Omron Sysmac Studio project Auto Connect Project (Sysmac Studio 1.66.0.64007, StandardProject)

# Controller new_Controller_0: NX502-1300 version 1.69
Units and slaves: Node9 : CPX-AP-A-EC-M12(E007); 0 : CPX-AP-A-EC-M12(M1); 1 : CPX-AP-A-16DI-D-M12-5P(M2); 2 : CPX-AP-A-16DI-D-M12-5P(M3); 3 : VABX-A-P-EL-E12-APA(M4); Node10 : NXR-ILM08C-ECT (E006); Unit 1 : NX-PF0730 (N1); Unit 3 : NX-SID800 (N3); Unit 4 : NX-SID800 (N4); Unit 5 : NX-SID800 (N5); Unit 6 : NX-SOD400 (N6); Unit 7 : NX-SOD400 (N7); Unit 8 : NX-PD1000 (N8); Unit 9 : NX-ID5442 (N9); Unit 10 : NX-ID5442 (N10); Unit 11 : NX-OD5256 (N11); Unit 12 : NX-OD5256 (N12)
Axis SC1501Ax, settings changed from default: AxisType=ServoType, UnitsConversion=EnumElement2, UnitsNumerator=8388608, ReducerUse=EnumElement2, UnitsDenominator=12.5, TravelDistancePerWorkRotation=125, MotorGearRatio=7, MaxVelocity=3199, MaxJogVelocity=3199, HomingMode=BackupAndPressingTime, StartDirection=NegativeDirection, OriginInputDetectionDirection=NegativeDirection, HomingVelocity=20, HomingApproachVelocity=20, HomingAcceleration=10, HomingJerk=10, PushTime=0, CompensationVelocity=20, EncoderTypes=Abs
Axis SC2301Ax, settings changed from default: AxisNumber=1, AxisType=ServoType, UnitsConversion=EnumElement2, UnitsNumerator=8601600, UnitsDenominator=30.0372, TravelDistancePerWorkRotation=300.37, MotorGearRatio=10, MaxVelocity=7499, MaxJogVelocity=7499, MaxAcceleration=10000, MaxDeceleration=10000, FollowingErrorLimit=500, FollowingErrorAlarmLimit=500, HomingMode=BackupAndPressingTime, HomingVelocity=10, HomingApproachVelocity=10, HomingAcceleration=50, HomingDeceleration=50, HomingJerk=100, PushTime=0
Axis SC2302Ax, settings changed from default: AxisNumber=2, AxisType=ServoType, UnitsConversion=EnumElement2, UnitsNumerator=8388608, ReducerUse=EnumElement2, UnitsDenominator=30.0372, TravelDistancePerWorkRotation=300.37, MotorGearRatio=10, MaxVelocity=7499, MaxJogVelocity=7499, MaxAcceleration=10000, MaxDeceleration=10000, FollowingErrorLimit=500, FollowingErrorAlarmLimit=500, HomingMode=BackupAndPressingTime, StartDirection=NegativeDirection, OriginInputDetectionDirection=NegativeDirection, HomingVelocity=10, HomingApproachVelocity=10, HomingAcceleration=50, HomingDeceleration=50, HomingJerk=50, PushTime=0
Axis SC2303Ax, settings changed from default: AxisNumber=3, AxisType=ServoType, UnitsConversion=EnumElement2, UnitsNumerator=8388608, ReducerUse=EnumElement2, UnitsDenominator=30.0372, TravelDistancePerWorkRotation=300.37, MotorGearRatio=10, MaxVelocity=7499, MaxJogVelocity=7499, MaxAcceleration=10000, MaxDeceleration=10000, FollowingErrorLimit=500, FollowingErrorAlarmLimit=500, HomingMode=BackupAndPressingTime, StartDirection=NegativeDirection, OriginInputDetectionDirection=NegativeDirection, HomingVelocity=10, HomingApproachVelocity=10, HomingAcceleration=50, HomingJerk=50, PushTime=0
Axis SC6401Ax, settings changed from default: AxisNumber=4, AxisType=ServoType, UnitsConversion=EnumElement2, UnitsNumerator=8388608, ReducerUse=EnumElement2, UnitsDenominator=9, TravelDistancePerWorkRotation=125, MotorGearRatio=10, MaxVelocity=2299, MaxJogVelocity=2299, HomingMode=BackupAndProximitySignalOn, StartDirection=NegativeDirection, OriginInputDetectionDirection=NegativeDirection, HomingVelocity=20, HomingApproachVelocity=20, EncoderTypes=Abs
Task PrimaryTask (priority 4, period or condition 4000): Control, Inputs, Outputs
Library OneS_monitor 1.0.0 (contents left out)

TYPE CylinderD : STRUCT
    AutoExtend : BOOL;
    AutoRetract : BOOL;
    ManExtend : BOOL;
    ManRetract : BOOL;
    ManOff : BOOL;
    ForceExtend : BOOL;
    ForceRetract : BOOL;
    ExtendSol : BOOL;
    RetractSol : BOOL;
    TestCycleSelect : BOOL;
    AlarmMute : BOOL;
    ExtendReed : BOOL;
    RetractReed : BOOL;
    Alarm : BOOL;
    CountReset : BOOL;
    CycleExtendTime : LREAL;
    CycleRetractTime : LREAL;
    ExtendTime : LREAL;
    RetractTime : LREAL;
    ExtendTimeAcc : LREAL;
    RetractTimeAcc : LREAL;
    AlarmCode : DINT;
    ManualCode : DINT;
    ExtendReedsUsed : DINT;
    RetractReedsUsed : DINT;
    ExtendCount : DINT;
    RetractCount : DINT;
    TagName : STRING[256];
    TagDescription : STRING[256];
    ErrorTrigger : ARRAY[0..19] OF BOOL;
    ManualTrigger : ARRAY[0..19] OF BOOL;
END_STRUCT END_TYPE
TYPE MotorD : STRUCT
    AlarmMute : BOOL;
    AutoForward : BOOL;
    ManForward : BOOL;
    ManReverse : BOOL;
    ManOFF : BOOL;
    AutoReverse : BOOL;
    ForceFoward : BOOL;
    ForceReverse : BOOL;
    RunFeedback : BOOL;
    Alarm : BOOL;
    ForceOFF : BOOL;
    CountReset : BOOL;
    ManualCode : DINT;
    AlarmCode : DINT;
    RunCount : DINT;
    RunHours : REAL;
    Faulttime : LREAL;
    FaulttimeAcc : LREAL;
    TagName : STRING[256];
    TagDescription : STRING[256];
    ErrorTrigger : ARRAY[0..19] OF BOOL;
    ManualTrigger : ARRAY[0..19] OF BOOL;
END_STRUCT END_TYPE
TYPE MotorVSDD : STRUCT
    AlarmMute : BOOL;
    AutoForward : BOOL;
    ManForward : BOOL;
    ManReverse : BOOL;
    ManOFF : BOOL;
    AutoReverse : BOOL;
    ForceFoward : BOOL;
    ForceReverse : BOOL;
    ForceOFF : BOOL;
    CountReset : BOOL;
    RunFeedback : BOOL;
    ManualCode : DINT;
    AlarmCode : DINT;
    RunCount : DINT;
    RunHours : REAL;
    Faulttime : LREAL;
    FaulttimeAcc : LREAL;
    AutoSpeed : UINT;
    ManualSpeed : UINT;
    Speed : UINT;
    Alarm : BOOL;
    TagName : STRING[256];
    TagDescription : STRING[256];
    ErrorTrigger : ARRAY[0..19] OF BOOL;
    ManualTrigger : ARRAY[0..19] OF BOOL;
END_STRUCT END_TYPE
TYPE ServoD : STRUCT
    JogForward : BOOL;
    JogReverse : BOOL;
    JogToPosition : BOOL;
    ManualHome : BOOL;
    AutoHome : BOOL;
    Homed : BOOL;
    Alarm : BOOL;
    Enabled : BOOL;
    AxisErrorCode : WORD;
    RunHours : REAL;
    JogSpeed : LREAL;
    JogAccel : LREAL;
    JogDecel : LREAL;
    JogPos : LREAL;
    JogJerk : LREAL;
    JogType : DINT;
    ActualPos : LREAL;
    ActualVel : LREAL;
    PowerEnable : BOOL;
    MovePos1 : BOOL;
    Pos1 : LREAL;
    Pos1Vel : LREAL;
    Pos1Accel : LREAL;
    Pos1Decel : LREAL;
    Pos1Jerk : LREAL;
    Pos1Movetype : DINT;
    Pos1OK : BOOL;
    MovePos2 : BOOL;
    Pos2 : LREAL;
    Pos2Vel : LREAL;
    Pos2Accel : LREAL;
    Pos2Decel : LREAL;
    Pos2Jerk : LREAL;
    Pos2Movetype : DINT;
    Pos2OK : BOOL;
    MovePos3 : BOOL;
    Pos3 : LREAL;
    Pos3Vel : LREAL;
    Pos3Accel : LREAL;
    Pos3Decel : LREAL;
    Pos3Jerk : LREAL;
    Pos3Movetype : DINT;
    Pos3OK : BOOL;
    MovePos4 : BOOL;
    Pos4 : LREAL;
    Pos4Vel : LREAL;
    Pos4Accel : LREAL;
    Pos4Decel : LREAL;
    Pos4Jerk : LREAL;
    Pos4OK : BOOL;
    Pos4Movetype : DINT;
    MovePos5 : BOOL;
    Pos5 : LREAL;
    Pos5Vel : LREAL;
    Pos5Accel : LREAL;
    Pos5Decel : LREAL;
    Pos5OK : BOOL;
    Pos5Movetype : DINT;
    Pos5Jerk : LREAL;
    MoveVelSpeed : LREAL;
    MovePos6 : BOOL;
    Pos6 : LREAL;
    Pos6Vel : LREAL;
    Pos6Accel : LREAL;
    Pos6Decel : LREAL;
    Pos6Jerk : LREAL;
    Pos6OK : BOOL;
    Pos6Movetype : DINT;
    MoveVel : BOOL;
    MoveVelAcc : LREAL;
    MoveVeldec : LREAL;
    MoveVelJerk : LREAL;
    MoveVelType : DINT;
    MoveVelCon : BOOL;
    MoveVelOK : BOOL;
    PositionTolerence : LREAL;
    AlarmCode : DWORD;
    ManualCode : DINT;
    TagName : STRING[256];
    TagDescription : STRING[256];
    ErrorTrigger : ARRAY[0..19] OF BOOL;
    ManualTrigger : ARRAY[0..19] OF BOOL;
END_STRUCT END_TYPE
TYPE MiscInD : STRUCT
    ManOn : BOOL;
    ManOff : BOOL;
    ForceOn : BOOL;
    ForceOff : BOOL;
    Fault : BOOL;
    InputFault : BOOL;
    Mute : BOOL;
    Value : BOOL;
    Input : BOOL;
    AlarmCode : DINT;
    Alarm : BOOL;
    ManualCode : DINT;
    DebounceOFFtime : LREAL;
    DebounceONtime : LREAL;
    FaultTime : LREAL;
    AccumulatedOnTime : LREAL;
    AccumulatedOffTime : LREAL;
    FaultAccumulatedTime : LREAL;
    TagName : STRING[256];
    TagDescription : STRING[256];
    ErrorTrigger : ARRAY[0..19] OF BOOL;
    ManualTrigger : ARRAY[0..19] OF BOOL;
END_STRUCT END_TYPE
TYPE MiscOutD : STRUCT
    ManOn : BOOL;
    ManOff : BOOL;
    ForceOn : BOOL;
    ForceOff : BOOL;
    Fault : BOOL;
    Mute : BOOL;
    Value : BOOL;
    Auto : BOOL;
    AlarmCode : DINT;
    ManualCode : DINT;
    FaultTime : LREAL;
    FaultAccumulatedTime : LREAL;
    Alarm : BOOL;
    TagName : STRING[256];
    TagDescription : STRING[256];
    ErrorTrigger : ARRAY[0..19] OF BOOL;
    ManualTrigger : ARRAY[0..19] OF BOOL;
END_STRUCT END_TYPE
TYPE SequenceD : STRUCT
    CurrentStep : ARRAY[0..31] OF BOOL;
    StepTime : ARRAY[0..31] OF REAL;
    StepTimeAcc : REAL;
    Matrix : ARRAY[0..31] OF Dint_Bool;
    Matrix_In : ARRAY[0..31] OF DINT;
    Outputs : ARRAY[0..0] OF Dint_Bool;
    StepReq : DINT;
    StepNum : DINT;
    StepPrev : DINT;
    LastActiveStep : DINT;
    StepTimeDn : BOOL;
    History : ARRAY[0..9] OF SequenceHistory;
    SequenceDisabled : BOOL;
    TagName : STRING[256];
    TagDiscription : STRING[256];
    LocalMessageOffset : DINT;
    LocalMessageValue : DINT;
    Flag : ARRAY[0..9] OF BOOL;
    DeviceAlarm : BOOL;
    Held : BOOL;
    Stopped : BOOL;
    Homed : BOOL;
    TagName_Copy : STRING[256];
    TagDescription : STRING[256];
END_STRUCT END_TYPE
TYPE SequenceHistory : STRUCT
    Num : DINT;
    Messageoffset : DINT;
    ElapsedTime : REAL;
END_STRUCT END_TYPE
TYPE System : STRUCT
    ScanRate : REAL;
    Alarm : BOOL;
    Alarm_Ack : BOOL;
    Energized : BOOL;
    Safetyresetselect : BOOL;
    CurrentStep : DINT;
    ResetSelect : BOOL;
    Messages : DINT;
    AlertMessages : DINT;
    SafetyMessages : DINT;
    HomeSelect : BOOL;
    HomeEnabled : BOOL;
    Homed : BOOL;
    StartSelect : BOOL;
    HoldSelect : BOOL;
    Alarm_AckSelect : BOOL;
    StopSelect : BOOL;
    Alert : BOOL;
    CycleTime : LREAL;
    ShippersPerMin : LREAL;
    TotalRunHours : LREAL;
    CartonsPerMin : LREAL;
END_STRUCT END_TYPE
TYPE TrackTrace : STRUCT
    Carton : DINT;
    Booklet : BOOL;
END_STRUCT END_TYPE
TYPE Vis_In : STRUCT
    InfoBits : SINT;
    Reserved1 : SINT;
    Congiguration_change_device : SINT;
    Reserved2 : BYTE;
    Device_Status : Device_status;
    Fault_code : DINT;
    Counters : ARRAY[0..5] OF DINT;
    Read_Cyc_report : ARRAY[0..3] OF int;
    Decode_Cyc_report : ARRAY[0..3] OF int;
    CodeType : DINT;
    PixelPerElement : real;
    Decode_length : DINT;
    Decode_data : ARRAY[0..435] OF Byte;
END_STRUCT END_TYPE
TYPE Device_status : STRUCT
    Run_mode : BOOL;  (* offset 0.0 *)
    Triger_Acknowledged : BOOL;  (* offset 0.1 *)
    Exposure_done : BOOL;  (* offset 0.2 *)
    Decoding : BOOL;  (* offset 0.3 *)
    Data_is_Ready : BOOL;  (* offset 0.4 *)
    Read_cyc_pass : BOOL;  (* offset 0.5 *)
    Read_cyc_fail : BOOL;  (* offset 0.6 *)
    General_Fault : BOOL;  (* offset 0.7 *)
    New_match_code_acknowledged : BOOL;  (* offset 1.0 *)
    Match_code_enabled : BOOL;  (* offset 1.1 *)
    Image_sensor_Calibrating : BOOL;  (* offset 1.2 *)
    Image_sensor_Calibrating_complete : BOOL;  (* offset 1.3 *)
    Training : BOOL;  (* offset 1.4 *)
    Training_complete : BOOL;  (* offset 1.5 *)
    Optimizing_complete : BOOL;  (* offset 1.6 *)
    Auto_image_photometry_enabled : BOOL;  (* offset 1.7 *)
    Auto_image_photometry_Complete : BOOL;  (* offset 2.0 *)
    Output1_Status : BOOL;  (* offset 2.1 *)
    Output2_Status : BOOL;  (* offset 2.2 *)
    Output3_Status : BOOL;  (* offset 2.3 *)
    Buffer_overflow : BOOL;  (* offset 2.4 *)
    Reserved : ARRAY[0..9] OF Bool;  (* offset 2.5 *)
END_STRUCT END_TYPE
TYPE Vis_out : STRUCT
    Command : commands;
END_STRUCT END_TYPE
TYPE commands : STRUCT
    Run_mode : BOOL;  (* offset 0.0 *)
    Trigger : BOOL;  (* offset 0.1 *)
    Enable_match_code : BOOL;  (* offset 0.2 *)
    Reset_general_fault : BOOL;  (* offset 0.3 *)
    Clear_NoRead_CycRead_Count : BOOL;  (* offset 0.4 *)
    Clear_Mismatch_CycRead_Count : BOOL;  (* offset 0.5 *)
    Clear_NoRead_Count : BOOL;  (* offset 0.6 *)
    Clear_trigger_Count : BOOL;  (* offset 0.7 *)
    Clear_MatchCode_count : BOOL;  (* offset 1.0 *)
    Clear_Mismatch_Count : BOOL;  (* offset 1.1 *)
    Output_1 : BOOL;  (* offset 1.2 *)
    Output_2 : BOOL;  (* offset 1.3 *)
    Output_3 : BOOL;  (* offset 1.4 *)
    Reserved : ARRAY[0..17] OF Bool;  (* offset 1.5 *)
END_STRUCT END_TYPE
TYPE Resulted : STRUCT
    ScanData : STRING[32];
    Done : BOOL;
    Match : BOOL;
    Mismatch : BOOL;
    Alarm : BOOL;
END_STRUCT END_TYPE
TYPE ScannerD : STRUCT
    Result : Resulted;
    ExpectedCode : STRING[32];
    Trigger : BOOL;
    Alarm : BOOL;
    AlarmMute : BOOL;
    AlarmCode : DINT;
END_STRUCT END_TYPE
TYPE BatchDetails : STRUCT
    Start : BOOL;  (* Batch Start *)
    Running : BOOL;  (* Running *)
    Innitiate : BOOL;  (* Innitialization *)
    Complete : BOOL;  (* Batch Complete *)
    Goodshippers : REAL;  (* Good shipper *)
    Rejectshippers : REAL;  (* Reject shipper *)
    Totalshippers : REAL;  (* Total shipper *)
END_STRUCT END_TYPE
TYPE RecipeD : STRUCT
    RealValue : ARRAY[0..49] OF REAL;
    MechValue : ARRAY[0..49] OF REAL;
END_STRUCT END_TYPE
TYPE Word_Bool : UNION
    Word_value : Word;
    Bool_value : ARRAY[0..31] OF BOOL;
END_UNION END_TYPE
TYPE Dint_Bool : UNION
    Dint_Value : DWORD;
    Bool_Value : ARRAY[0..31] OF BOOL;
END_UNION END_TYPE

VAR_GLOBAL RETAIN
    CY1601 : CylinderD;  (* Shipper Support Cylinder; published *)
    PE1404 : MiscInD;  (* published *)
    CY2502 : CylinderD;  (* Product Clamp CYL 2; published *)
    CY2501 : CylinderD;  (* Vertical CYL 1; published *)
    CY2402 : CylinderD;  (* Vertical Stopper CYL; published *)
    CY2401 : CylinderD;  (* Matrix Pusher CYL; published *)
    CY2302 : CylinderD;  (* Matrix Side Shift Cyl 1 at matrix area 2; published *)
    CY2303 : CylinderD;  (* Bottles stopper Cyl 1 @ area 1; RetractReed Bottles stopper Cyl 1 @ area 1; published *)
    CY2301 : CylinderD;  (* Matrix Side Shift Cyl 1 at matrix area 1; published *)
    PE1501 : MiscInD;  (* Shipper Presence Detect; Value Plucker Head Shipper Presence Detect; published *)
    PE2201 : MiscInD;  (* Shipper Squaring Detect PE; published *)
    PE2202 : MiscInD;  (* Bottom tape Low level Detect; published *)
    PE2203 : MiscInD;  (* Bottom Tape apply Check PE 1; published *)
    PE2301 : MiscInD;  (* Matrix Present Detetct Eye1; published *)
    PE2302 : MiscInD;  (* Matrix Present Detetct Eye2; published *)
    PE2303 : MiscInD;  (* Product Presnt @ Collation Entrc; published *)
    PE2401 : MiscInD;  (* Matrix Present Detect; published *)
    PE3401 : MiscInD;  (* Pre-Lable Trigger PE; published *)
    PE3402 : MiscInD;  (* Shipper presence for Palletizer; published *)
    PE6901 : MiscInD;  (* Pallet 1 Presence PE 1; published *)
    PE6902 : MiscInD;  (* Pallet 1 Presence PE 2; published *)
    DI3511 : MiscInD;  (* Pre-Printing Applicator Machine Run Signal; published *)
    DI3501 : MiscInD;  (* Label Applicator Machine Run Signal; published *)
    DI3502 : MiscInD;  (* Label Applicator Machine Accept Signal; published *)
    DI3503 : MiscInD;  (* Label Applicator Machine Reject Signal; published *)
END_VAR
VAR_GLOBAL
    SC2701 : ServoD;  (* Shipper pusher Servo; published *)
END_VAR
VAR_GLOBAL RETAIN
    MO1402 : MotorD;  (* Magazine motor 2; published *)
    MO2301 : MotorD;  (* Infeed Collation Conveyor Motor; published *)
    MO2201 : MotorD;  (* Tapping Machine RH Motor; published *)
    MO2202 : MotorD;  (* Tapping Machine LH Motor; published *)
    IL0302 : MiscOutD;  (* Alert Indication (Amber); published *)
    IL0303 : MiscOutD;  (* Fault Indication (Red); published *)
    DO0301 : MiscOutD;  (* Drives Fault Reset; published *)
    DO3301 : MiscOutD;  (* Aggrigation System Trigger Signal; published *)
    DO3302 : MiscOutD;  (* published *)
    SV0401 : MiscOutD;  (* Pneumatic Quick Exhaust Valve; published *)
    SV1501 : MiscOutD;  (* Plucker Vacuum Sov 1; published *)
    SV2301 : MiscOutD;  (* Vaccume SOL; published *)
    SV2501 : MiscOutD;  (* Pickhead Vacuum Sov 1; published *)
    SV2502 : MiscOutD;  (* Pickhead Vacuum Sov 2; published *)
    PS2501 : MiscInD;  (* Robot pickhead pressure switch; published *)
    PS0401 : MiscInD;  (* Presure Switch; published *)
    IL0301 : MiscOutD;  (* Run Indication (Green); published *)
    P23c : SequenceD;  (* Infeed Conveyor 3; published *)
END_VAR
VAR_GLOBAL
    SafetyDeviceReady : BOOL;  (* Emergency and Guard Door Ready; published *)
END_VAR
VAR_GLOBAL RETAIN
    Batch_Report : BatchDetails;  (* published *)
END_VAR
VAR_GLOBAL
    Shipper_Accept : BOOL;
END_VAR
VAR_GLOBAL RETAIN
    CY2304 : CylinderD;  (* Bottles stopper Cyl 1 @ area 2; published *)
END_VAR
VAR_GLOBAL
    Reject_Matrix_Accept : BOOL;
    Carton_Matrix_Accept : BOOL;
    RO4001_I_PalletizingDone : BOOL;
    Palletizing_Done : BOOL;
    Shipper_Reject : BOOL;
    Shipper_Good_Count : BOOL;
    S_CellEnabled : BOOL;
    SKU_Select : DINT;
END_VAR
VAR_GLOBAL RETAIN
    P27 : SequenceD;  (* Case Erector; Flag[0] Plucker At Shipper Pick Pos; published *)
    PE1602 : MiscInD;  (* published *)
END_VAR
VAR_GLOBAL
    TotalLayers : DINT;  (* published *)
    ShippersPerLayer : DINT;  (* published *)
    IPCcheck : BOOL;  (* published *)
    IPCcheckAlarm : BOOL;
    IPCCheck1 : BOOL;  (* published *)
    P22_TapeAlarm : BOOL;  (* published *)
    RO4001_Alarm : BOOL;
    RO4001_ErrorTrigger : ARRAY[0..9] OF BOOL;  (* published *)
END_VAR
VAR_GLOBAL RETAIN
    DO3502 : MiscOutD;  (* published *)
    DO3501 : MiscOutD;  (* published *)
    PE3501 : MiscInD;  (* published *)
    K1301 : MiscOutD;  (* published *)
    PE1403 : MiscInD;  (* Shipper Forming Detect PE 2; published *)
    PE1402 : MiscInD;  (* Shipper Forming Detect PE 1; published *)
    SV2701 : MiscOutD;  (* published *)
    PE6401 : MiscInD;  (* Shipper Presence Detect Eye; published *)
    PE1801 : MiscInD;  (* Product High Level Detect; published *)
    PE1811 : MiscInD;  (* Bundle High level detect; published *)
    PE1812 : MiscInD;  (* Bundle detect @ Clamp; published *)
    PE1701 : MiscInD;  (* Shipper Presence @ Stopper 1; published *)
    PE1702 : MiscInD;  (* Shipper Presence @ Placing Station; published *)
    PE2501 : MiscInD;  (* published *)
    PE2502 : MiscInD;  (* published *)
    PE2503 : MiscInD;  (* published *)
    PE2801 : MiscInD;  (* Layer Board Magazine Low level detect Eye; published *)
    PE2511 : MiscInD;  (* published *)
    PE2521 : MiscInD;  (* published *)
    PE2702 : MiscInD;  (* published *)
    PE2703 : MiscInD;  (* published *)
END_VAR
VAR_GLOBAL
    PE7101 : MiscInD;  (* Shipper Presence Detect; published *)
END_VAR
VAR_GLOBAL RETAIN
    PE3101 : MiscInD;  (* published *)
    PE2512 : MiscInD;  (* published *)
    PE6911 : MiscInD;  (* published *)
    PE6912 : MiscInD;  (* published *)
    SV1502 : MiscOutD;  (* Plucker Vacuum Sov 1; published *)
    SV1503 : MiscOutD;  (* Plucker Vacuum Sov 1; published *)
    SV2511 : MiscOutD;  (* published *)
    SV2512 : MiscOutD;  (* published *)
    SV2521 : MiscOutD;  (* published *)
    SV7101 : MiscOutD;  (* Shipper Vaccume; published *)
    DO320 : MiscOutD;
    DO0320 : MiscOutD;
    DO0350 : MiscOutD;
    CY1502 : CylinderD;  (* Minor Flap close CYL 2; ExtendReed Minor Flap close CYL 2; published *)
    CY1503 : CylinderD;  (* Major Flap close CYL 1; RetractReed Major Flap close CYL 1; published *)
    CY1504 : CylinderD;  (* Major Flap close CYL 2; RetractReed Major Flap close CYL 1; published *)
    CY1811 : CylinderD;  (* Clamp Cyl 1; published *)
    CY1701 : CylinderD;  (* Shipper Stopper Before Loading station.; published *)
    CY1702 : CylinderD;  (* Shipper Stopper at Loading station.; published *)
    CY1703 : CylinderD;  (* Hopper Cylinder; published *)
    CY2521 : CylinderD;  (* published *)
    CY7101 : CylinderD;  (* Shipper Rotation CYL; published *)
    CY7102 : CylinderD;  (* Shipper Puller and Pusher CYL; published *)
    CY3401 : CylinderD;  (* Shipper Stopper CYL; published *)
    CY3402 : CylinderD;  (* Shipper Rejection/ Accepted CYL; published *)
    DI0350 : MiscInD;  (* published *)
    DI7501 : MiscInD;  (* published *)
    DI7502 : MiscInD;  (* published *)
    DI7503 : MiscInD;  (* published *)
    DI3512 : MiscInD;  (* published *)
    DI3513 : MiscInD;  (* published *)
    MO1801 : MotorD;  (* Infeed Conveyor 1 of Loose Bottles Motor; published *)
    MO1811 : MotorD;  (* Infeed Conveyor 2 of Bundle Bottles Motor; published *)
    MO1701 : MotorD;  (* Main Drive Conveyor Motor; published *)
    MO3101 : MotorD;  (* published *)
    SC1501 : ServoD;  (* Plucker Servo; published *)
END_VAR
VAR_GLOBAL
    SC1501_Ax : _sAXIS_REF;
END_VAR
VAR_GLOBAL RETAIN
    SC6401 : ServoD;  (* Box Transfer Servo; published *)
END_VAR
VAR_GLOBAL
    SC6401_Ax : _sAXIS_REF;
END_VAR
VAR_GLOBAL RETAIN
    SC2301 : ServoD;  (* published *)
END_VAR
VAR_GLOBAL
    SC2301_Ax : _sAXIS_REF;
END_VAR
VAR_GLOBAL RETAIN
    SC2302 : ServoD;  (* published *)
END_VAR
VAR_GLOBAL
    SC2302_Ax : _sAXIS_REF;
END_VAR
VAR_GLOBAL RETAIN
    SC2303 : ServoD;  (* published *)
END_VAR
VAR_GLOBAL
    SC2303_Ax : _sAXIS_REF;
    XC0301_6_I : ARRAY[0..15] OF BOOL;  (* Input Card 1; at IOBus://unit#9/Input Bit 16 bits *)
    XC0301_7_I : ARRAY[0..15] OF BOOL;  (* Input Card 2; at IOBus://unit#10/Input Bit 16 bits *)
END_VAR
VAR_GLOBAL RETAIN
    PS2502 : MiscInD;  (* published *)
END_VAR
VAR_GLOBAL
    XC0301_8_O : ARRAY[0..15] OF BOol;  (* Output Card 1; at IOBus://unit#11/Output Bit 16 bits *)
END_VAR
VAR_GLOBAL RETAIN
    IL0304 : MiscOutD;  (* Buzzer; published *)
END_VAR
VAR_GLOBAL
    XC0301_9_O : ARRAY[0..15] OF BOOL;  (* Output Card 2; at IOBus://unit#12/Output Bit 16 bits *)
    A0XC0401_1_I_0 : BOOL;  (* at ECAT://node#[9,1]/Inputs_Input 0_6000_01 *)
    A0XC0401_1_I_1 : BOOL;  (* at ECAT://node#[9,1]/Inputs_Input 1_6000_02 *)
    A0XC0401_1_I_3 : BOOL;  (* at ECAT://node#[9,1]/Inputs_Input 3_6000_04 *)
    A0XC0401_1_I_4 : BOOL;  (* at ECAT://node#[9,1]/Inputs_Input 4_6000_05 *)
    A0XC0401_1_I_5 : BOOL;  (* at ECAT://node#[9,1]/Inputs_Input 5_6000_06 *)
    A0XC0401_1_I_6 : BOOL;  (* at ECAT://node#[9,1]/Inputs_Input 6_6000_07 *)
    A0XC0401_1_I_7 : BOOL;  (* at ECAT://node#[9,1]/Inputs_Input 7_6000_08 *)
    A0XC0401_1_I_8 : BOOL;  (* at ECAT://node#[9,1]/Inputs_Input 8_6000_09 *)
    A0XC0401_1_I_9 : BOOL;  (* at ECAT://node#[9,1]/Inputs_Input 9_6000_0A *)
    A0XC0401_1_I_10 : BOOL;  (* at ECAT://node#[9,1]/Inputs_Input 10_6000_0B *)
    A0XC0401_1_I_11 : BOOL;  (* at ECAT://node#[9,1]/Inputs_Input 11_6000_0C *)
    A0XC0401_1_I_12 : BOOL;  (* at ECAT://node#[9,1]/Inputs_Input 12_6000_0D *)
    A0XC0401_1_O_8 : BOOL;
    A0XC0401_1_O_9 : BOOL;
    A0XC0401_1_O_10 : BOOL;
    A0XC0401_1_O_11 : BOOL;
    A0XC0401_1_O_12 : BOOL;
    A0XC0401_1_O_13 : BOOL;
    XC0320_1_I_0 : BOOL;  (* Remote I/O Link Collation Pickhead; at ECAT://node#10/Port1 Input Data01/Port1 Port1 Pin4 Input Bit *)
    A0XC0401_1_O_0 : BOOL;  (* at ECAT://node#[9,3]/Outputs_Coil 0_7000_01 *)
    A0XC0401_1_O_1 : BOOL;  (* at ECAT://node#[9,3]/Outputs_Coil 1_7000_02 *)
    A0XC0401_1_O_2 : BOOL;  (* at ECAT://node#[9,3]/Outputs_Coil 2_7000_03 *)
    A0XC0401_1_O_3 : BOOL;  (* at ECAT://node#[9,3]/Outputs_Coil 3_7000_04 *)
    A0XC0401_1_O_4 : BOOL;  (* at ECAT://node#[9,3]/Outputs_Coil 4_7000_05 *)
    A0XC0401_1_O_5 : BOOL;  (* at ECAT://node#[9,3]/Outputs_Coil 5_7000_06 *)
    A0XC0401_1_O_6 : BOOL;  (* at ECAT://node#[9,3]/Outputs_Coil 6_7000_07 *)
    A0XC0401_1_O_7 : BOOL;  (* at ECAT://node#[9,3]/Outputs_Coil 7_7000_08 *)
    A0XC0401_2_O_0 : BOOL;  (* at ECAT://node#[9,3]/Outputs_Coil 8_7000_09 *)
    A0XC0401_2_O_1 : BOOL;  (* at ECAT://node#[9,3]/Outputs_Coil 9_7000_0A *)
    A0XC0401_2_O_2 : BOOL;  (* at ECAT://node#[9,3]/Outputs_Coil 10_7000_0B *)
    A0XC0401_2_O_3 : BOOL;  (* at ECAT://node#[9,3]/Outputs_Coil 11_7000_0C *)
    A0XC0401_2_O_4 : BOOL;  (* at ECAT://node#[9,3]/Outputs_Coil 12_7000_0D *)
    A0XC0401_2_O_5 : BOOL;  (* at ECAT://node#[9,3]/Outputs_Coil 13_7000_0E *)
    A0XC0401_2_O_6 : BOOL;  (* at ECAT://node#[9,3]/Outputs_Coil 14_7000_0F *)
    A0XC0401_2_O_7 : BOOL;  (* at ECAT://node#[9,3]/Outputs_Coil 15_7000_10 *)
    A0XC0401_3_O_0 : BOOL;  (* at ECAT://node#[9,3]/Outputs_Coil 16_7000_11 *)
    A0XC0401_3_O_1 : BOOL;  (* at ECAT://node#[9,3]/Outputs_Coil 17_7000_12 *)
    A0XC0401_3_O_2 : BOOL;  (* at ECAT://node#[9,3]/Outputs_Coil 18_7000_13 *)
    A0XC0401_3_O_3 : BOOL;  (* at ECAT://node#[9,3]/Outputs_Coil 19_7000_14 *)
    A0XC0401_3_O_4 : BOOL;  (* at ECAT://node#[9,3]/Outputs_Coil 20_7000_15 *)
    A0XC0401_3_O_5 : BOOL;  (* at ECAT://node#[9,3]/Outputs_Coil 21_7000_16 *)
    A0XC0401_3_O_6 : BOOL;  (* at ECAT://node#[9,3]/Outputs_Coil 22_7000_17 *)
    A0XC0401_3_O_7 : BOOL;  (* at ECAT://node#[9,3]/Outputs_Coil 23_7000_18 *)
    XC0320_1_I_1 : BOOL;  (* Remote I/O Link Collation Pickhead; at ECAT://node#10/Port1 Input Data01/Port1 Port1 Pin2 Input Bit *)
    XC0320_1_O_2 : BOOL;  (* Remote I/O Link Collation Pickhead *)
    XC0320_1_O_3 : BOOL;  (* Remote I/O Link Collation Pickhead *)
    XC0320_1_O_4 : BOOL;  (* Remote I/O Link Collation Pickhead *)
    XC0320_1_I_5 : BOOL;  (* Remote I/O Link Collation Pickhead; at ECAT://node#10/Port1 Input Data01/Port1 Port3 Pin2 Input Bit *)
    XC0320_1_I_6 : BOOL;  (* Remote I/O Link Collation Pickhead; at ECAT://node#10/Port1 Input Data01/Port1 Port4 Pin4 Input Bit *)
    XC0320_1_I_7 : BOOL;  (* Remote I/O Link Collation Pickhead; at ECAT://node#10/Port1 Input Data01/Port1 Port4 Pin2 Input Bit *)
    XC0320_1_I_8 : BOOL;  (* Remote I/O Link Collation Pickhead; at ECAT://node#10/Port1 Input Data01/Port1 Port5 Pin4 Input Bit *)
    XC0320_1_I_9 : BOOL;  (* Remote I/O Link Collation Pickhead; at ECAT://node#10/Port1 Input Data01/Port1 Port5 Pin2 Input Bit *)
    XC0320_1_I_10 : BOOL;  (* Remote I/O Link Collation Pickhead; at ECAT://node#10/Port1 Input Data01/Port1 Port6 Pin4 Input Bit *)
    XC0320_1_I_11 : BOOL;  (* Remote I/O Link Collation Pickhead; at ECAT://node#10/Port1 Input Data01/Port1 Port6 Pin2 Input Bit *)
    XC0320_1_I_12 : BOOL;  (* Remote I/O Link Collation Pickhead; at ECAT://node#10/Port1 Input Data01/Port1 Port7 Pin4 Input Bit *)
    XC0320_1_I_13 : BOOL;  (* Remote I/O Link Collation Pickhead; at ECAT://node#10/Port1 Input Data01/Port1 Port7 Pin2 Input Bit *)
    XC0320_1_I_14 : BOOL;  (* Remote I/O Link Collation Pickhead; at ECAT://node#10/Port1 Input Data01/Port1 Port8 Pin4 Input Bit *)
    XC0320_1_I_15 : BOOL;  (* Remote I/O Link Collation Pickhead; at ECAT://node#10/Port1 Input Data01/Port1 Port8 Pin2 Input Bit *)
    XC0320_2_O_0 : BOOL;  (* Remote I/O Link Rotary Roller *)
    XC0320_2_O_1 : BOOL;  (* Remote I/O Link Rotary Roller *)
    XC0320_2_O_2 : BOOL;  (* Remote I/O Link Rotary Roller *)
    XC0320_2_O_3 : BOOL;  (* Remote I/O Link Rotary Roller *)
    XC0320_2_O_4 : BOOL;  (* Remote I/O Link Rotary Roller *)
    XC0320_2_O_5 : BOOL;  (* Remote I/O Link Rotary Roller *)
    XC0320_2_O_6 : BOOL;  (* Remote I/O Link Rotary Roller *)
    XC0320_2_I_7 : BOOL;  (* Remote I/O Link Rotary Roller; at ECAT://node#10/Port2 Input Data01/Port2 Port4 Pin2 Input Bit *)
    XC0320_2_I_8 : BOOL;  (* Remote I/O Link Rotary Roller; at ECAT://node#10/Port2 Input Data01/Port2 Port5 Pin4 Input Bit *)
    XC0320_2_I_9 : BOOL;  (* Remote I/O Link Rotary Roller; at ECAT://node#10/Port2 Input Data01/Port2 Port5 Pin2 Input Bit *)
    XC0320_2_I_10 : BOOL;  (* Remote I/O Link Rotary Roller; at ECAT://node#10/Port2 Input Data01/Port2 Port6 Pin4 Input Bit *)
    XC0320_2_I_11 : BOOL;  (* Remote I/O Link Rotary Roller; at ECAT://node#10/Port2 Input Data01/Port2 Port6 Pin2 Input Bit *)
    XC0320_2_I_12 : BOOL;  (* Remote I/O Link Rotary Roller; at ECAT://node#10/Port2 Input Data01/Port2 Port7 Pin4 Input Bit *)
    XC0320_2_I_13 : BOOL;  (* Remote I/O Link Rotary Roller; at ECAT://node#10/Port2 Input Data01/Port2 Port7 Pin2 Input Bit *)
    XC0320_2_I_14 : BOOL;  (* Remote I/O Link Rotary Roller; at ECAT://node#10/Port2 Input Data01/Port2 Port8 Pin4 Input Bit *)
    XC0320_2_I_15 : BOOL;  (* Remote I/O Link Rotary Roller; at ECAT://node#10/Port2 Input Data01/Port2 Port8 Pin2 Input Bit *)
    XC0320_3_O_0 : BOOL;  (* Remote I/O Link Palletizer Robot , Labelling Conveyor, Pre Lable Applicator *)
    XC0320_3_O_1 : BOOL;  (* Remote I/O Link Palletizer Robot , Labelling Conveyor, Pre Lable Applicator *)
    XC0320_3_O_2 : BOOL;  (* Remote I/O Link Palletizer Robot , Labelling Conveyor, Pre Lable Applicator *)
    XC0320_3_O_3 : BOOL;  (* Remote I/O Link Palletizer Robot , Labelling Conveyor, Pre Lable Applicator *)
    XC0320_3_I_4 : BOOL;  (* Remote I/O Link Palletizer Robot , Labelling Conveyor, Pre Lable Applicator *)
    XC0320_3_I_5 : BOOL;  (* Remote I/O Link Palletizer Robot , Labelling Conveyor, Pre Lable Applicator *)
    XC0320_3_I_6 : BOOL;  (* Remote I/O Link Palletizer Robot , Labelling Conveyor, Pre Lable Applicator *)
    XC0320_3_I_7 : BOOL;  (* Remote I/O Link Palletizer Robot , Labelling Conveyor, Pre Lable Applicator *)
    XC0320_3_I_8 : BOOL;  (* Remote I/O Link Palletizer Robot , Labelling Conveyor, Pre Lable Applicator *)
    XC0320_3_I_9 : BOOL;  (* Remote I/O Link Palletizer Robot , Labelling Conveyor, Pre Lable Applicator *)
    XC0320_3_I_10 : BOOL;  (* Remote I/O Link Palletizer Robot , Labelling Conveyor, Pre Lable Applicator *)
    XC0320_3_I_11 : BOOL;  (* Remote I/O Link Palletizer Robot , Labelling Conveyor, Pre Lable Applicator *)
    XC0320_3_I_12 : BOOL;  (* Remote I/O Link Palletizer Robot , Labelling Conveyor, Pre Lable Applicator *)
    XC0320_3_I_13 : BOOL;  (* Remote I/O Link Palletizer Robot , Labelling Conveyor, Pre Lable Applicator *)
    XC0320_3_I_14 : BOOL;  (* Remote I/O Link Palletizer Robot , Labelling Conveyor, Pre Lable Applicator *)
    XC0320_3_I_15 : BOOL;  (* Remote I/O Link Palletizer Robot , Labelling Conveyor, Pre Lable Applicator *)
    XC0320_4_I_0 : BOOL;  (* Remote I/O Link Plucker; at ECAT://node#10/Port4 Input Data01/Port4 Port1 Pin4 Input Bit *)
    XC0320_4_I_1 : BOOL;  (* Remote I/O Link Plucker; at ECAT://node#10/Port4 Input Data01/Port4 Port1 Pin2 Input Bit *)
    XC0320_4_I_2 : BOOL;  (* Remote I/O Link Plucker; at ECAT://node#10/Port4 Input Data01/Port4 Port2 Pin4 Input Bit *)
    XC0320_4_I_3 : BOOL;  (* Remote I/O Link Plucker; at ECAT://node#10/Port4 Input Data01/Port4 Port2 Pin2 Input Bit *)
    XC0320_4_I_4 : BOOL;  (* Remote I/O Link Plucker; at ECAT://node#10/Port4 Input Data01/Port4 Port3 Pin4 Input Bit *)
    XC0320_4_I_5 : BOOL;  (* Remote I/O Link Plucker; at ECAT://node#10/Port4 Input Data01/Port4 Port3 Pin2 Input Bit *)
    XC0320_4_I_6 : BOOL;  (* Remote I/O Link Plucker; at ECAT://node#10/Port4 Input Data01/Port4 Port4 Pin4 Input Bit *)
    XC0320_4_I_7 : BOOL;  (* Remote I/O Link Plucker; at ECAT://node#10/Port4 Input Data01/Port4 Port4 Pin2 Input Bit *)
    XC0320_4_I_8 : BOOL;  (* Remote I/O Link Plucker; at ECAT://node#10/Port4 Input Data01/Port4 Port5 Pin4 Input Bit *)
    XC0320_4_I_9 : BOOL;  (* Remote I/O Link Plucker; at ECAT://node#10/Port4 Input Data01/Port4 Port5 Pin2 Input Bit *)
    XC0320_4_I_10 : BOOL;  (* Remote I/O Link Plucker; at ECAT://node#10/Port4 Input Data01/Port4 Port6 Pin4 Input Bit *)
    XC0320_4_I_11 : BOOL;  (* Remote I/O Link Plucker; at ECAT://node#10/Port4 Input Data01/Port4 Port6 Pin2 Input Bit *)
    XC0320_4_I_12 : BOOL;  (* Remote I/O Link Plucker; at ECAT://node#10/Port4 Input Data01/Port4 Port7 Pin4 Input Bit *)
    XC0320_4_I_13 : BOOL;  (* Remote I/O Link Plucker; at ECAT://node#10/Port4 Input Data01/Port4 Port7 Pin2 Input Bit *)
    XC0320_4_I_14 : BOOL;  (* Remote I/O Link Plucker; at ECAT://node#10/Port4 Input Data01/Port4 Port8 Pin4 Input Bit *)
    XC0320_4_I_15 : BOOL;  (* Remote I/O Link Plucker; at ECAT://node#10/Port4 Input Data01/Port4 Port8 Pin2 Input Bit *)
    XC0320_5_I_0 : BOOL;  (* Remote I/O Link Infeed Bundle & Main drive *)
    XC0320_5_I_1 : BOOL;  (* Remote I/O Link Infeed Bundle & Main drive *)
    XC0320_5_I_2 : BOOL;  (* Remote I/O Link Infeed Bundle & Main drive *)
    XC0320_5_I_3 : BOOL;  (* Remote I/O Link Infeed Bundle & Main drive *)
    XC0320_5_I_4 : BOOL;  (* Remote I/O Link Infeed Bundle & Main drive *)
    XC0320_5_I_5 : BOOL;  (* Remote I/O Link Infeed Bundle & Main drive *)
    XC0320_5_I_6 : BOOL;  (* Remote I/O Link Infeed Bundle & Main drive *)
    XC0320_5_I_7 : BOOL;  (* Remote I/O Link Infeed Bundle & Main drive *)
    XC0320_5_O_8 : BOOL;  (* Remote I/O Link Infeed Bundle & Main drive *)
    XC0320_5_O_9 : BOOL;  (* Remote I/O Link Infeed Bundle & Main drive *)
    XC0320_5_O_10 : BOOL;  (* Remote I/O Link Infeed Bundle & Main drive *)
    XC0320_5_I_11 : BOOL;  (* Remote I/O Link Infeed Bundle & Main drive *)
    XC0320_5_I_12 : BOOL;  (* Remote I/O Link Infeed Bundle & Main drive *)
    XC0320_5_I_13 : BOOL;  (* Remote I/O Link Infeed Bundle & Main drive *)
    XC0320_5_I_14 : BOOL;  (* Remote I/O Link Infeed Bundle & Main drive *)
    XC0320_5_I_15 : BOOL;  (* Remote I/O Link Infeed Bundle & Main drive *)
    DO3511 : MiscOutD;
END_VAR
VAR_GLOBAL RETAIN
    PE6903 : MiscInD;  (* Pallet 2 Presence PE 1; published *)
    PE6904 : MiscInD;  (* Pallet 2 Presence PE 2; published *)
END_VAR
VAR_GLOBAL
    A1_Control : System;  (* published *)
END_VAR
VAR_GLOBAL RETAIN
    PE1401 : MiscInD;  (* Magazine Low level detect Eye; Value Magazine Low level detect Eye; published *)
END_VAR
VAR_GLOBAL
    Zcomm : ARRAY[0..31] OF BOOL;
END_VAR
VAR_GLOBAL RETAIN
    PE2701 : MiscInD;  (* published *)
END_VAR
VAR_GLOBAL
    RESET_CMD : BOOL;  (* at IOBus://unit#2/RESET_CMD *)
    ES1001_I : BOOL;
    ES1201_I : BOOL;  (* at IOBus://unit#2/ES1201_I *)
    ES4001_I : BOOL;
    GZ1303_I : BOOL;  (* at IOBus://unit#2/GZ1303_I *)
    GZ1302_I : BOOL;  (* at IOBus://unit#2/GZ1302_I *)
END_VAR
VAR_GLOBAL RETAIN
    P22 : SequenceD;  (* P22 Step Engine; published *)
END_VAR
VAR_GLOBAL
    abc : INT;
    efd : INT;
    dsg : LREAL;
    CH : INT;
END_VAR
VAR_GLOBAL RETAIN
    Recipe : RecipeD;
    MO1401 : MotorD;  (* Magazine motor 1; published *)
    MO3401 : MotorD;  (* published *)
END_VAR
VAR_GLOBAL
    SKU_No : DINT;
END_VAR
VAR_GLOBAL RETAIN
    CY1501 : CylinderD;  (* Minor Flap close CYL 1; published *)
END_VAR
VAR_GLOBAL
    Ketan : WORD;
    Sandesh : WORD;
    jhsac : BOOL;
    ES1203_I : BOOL;  (* Emergency Switch 3; at IOBus://unit#2/ES1203_I *)
    ES1202_I : BOOL;  (* Emergency Switch 2; at IOBus://unit#2/ES1202_I; published *)
    GZ1304_I : BOOL;  (* Guard Door 4; at IOBus://unit#2/GZ1304_I; published *)
    GZ1305_I : BOOL;  (* Guard Door 5; at IOBus://unit#2/GZ1305_I; published *)
    GZ1301_I : BOOL;  (* Guard Door 1; at IOBus://unit#2/GZ1301_I; published *)
END_VAR
VAR_GLOBAL RETAIN
    P15 : SequenceD;  (* P15 Step Engine; Flag[0] Box Plucked Flag; Flag[1] Box Formed Flag; Flag[3] P15 Step Engine Box Plucked and Ready for box forming; published *)
    P64 : SequenceD;  (* P64 Step Engine; Flag[0] Box Transfer Assembly At Home Pos; Flag[1] Box Transferd Flag; Flag[2] P64 Step Engine Box Transfer Servo At Box Forming Pos; published *)
    P14 : SequenceD;  (* P14 Step Engine; Flag[0] Magzine_Ready_Flag; published *)
    P18 : SequenceD;  (* P18 Step Engine; Flag[2] Product Matrix Reday Flag To Collation Unit; published *)
    P18A : SequenceD;  (* P18a Step Engine; published *)
    P23 : SequenceD;  (* Flag[1] RO6302_Matrix_Pick_Flag; Flag[0] Collation_Unit_1_running; Flag[2] Collation_Unit_1_Complete; Flag[3] Colaation UNIT 1 Flag to Infeed COnveyor; published *)
    P17 : SequenceD;  (* P17 Step Engine; Flag[1] Main Drive Engine- Product Place Flag To ; published *)
    P28 : SequenceD;  (* P28 Step Engine *)
    P71 : SequenceD;  (* P71 Step Engine *)
    P23a : SequenceD;  (* Flag[0] Collation_Unit_2_Running; Flag[1] RO6302_Matrix_Pick_Flag; Flag[2] Collation_Unit_2_Complete *)
END_VAR
VAR_GLOBAL
    Collation_Unit_1_Define_RowsNo : REAL;  (* For Recipe HMI; published *)
    Collation_Unit_1_Running_RowsNo : INT;
END_VAR
VAR_GLOBAL RETAIN
    Product_Width : REAL;
END_VAR
VAR_GLOBAL
    SC2301_Pos2_Variable_1 : LREAL;
END_VAR
VAR_GLOBAL RETAIN
    SC2301_Pos2_Temp1 : REAL;
    SC2301_Pos2_Temp2 : REAL;
    SC2302_Pos2_Temp1 : REAL;
    SC2301_Pos3_Temp1 : REAL;
END_VAR
VAR_GLOBAL
    RO6301_Flag : BOOL;
END_VAR
VAR_GLOBAL RETAIN
    Collation_Unit_2_Define_RowsNo : REAL;
    SC2303_Pos2_Temp1 : REAL;
    SC2302_Pos4_Temp1 : REAL;
    Collation_Unit_1_Define_RowsNo_INT : INT;  (* Recipe Varibale *)
    Collation_Unit_2_Define_RowsNo_INT : INT;
END_VAR
VAR_GLOBAL
    RO6101_MatrixPlace : BOOL;
    RO6102_PartionPlace : BOOL;
END_VAR
VAR_GLOBAL RETAIN
    CY2305 : CylinderD;  (* published *)
    PE2204 : MiscInD;  (* published *)
    PE1703 : MiscInD;  (* published *)
    PE2206 : MiscInD;  (* published *)
    PE2205 : MiscInD;  (* published *)
END_VAR
VAR_GLOBAL
    ydytdutf : BOOL;
    ujcjgcj : BOOL;
    khvjk : BOOL;
    hkfvkhf : BOOL;
    PX1801 : MiscInD;  (* published *)
END_VAR
VAR_GLOBAL RETAIN
    MO2701 : MotorD;  (* Top Tapping Motor 1; published *)
    MO2702 : MotorD;  (* Top Tapping motor 2; published *)
    MO1802 : MotorD;  (* Lifting Conveyor; published *)
    SV2522 : MiscOutD;  (* published *)
END_VAR
VAR_GLOBAL
    CY2701 : CylinderD;
    A0XC0401_1_O_14 : BOOL;
    A0XC0401_1_O_15 : BOOL;
    A0XC0401_2_O_8 : BOOL;
    A0XC0401_2_O_9 : BOOL;
    A0XC0401_2_O_10 : BOOL;
    A0XC0401_2_O_11 : BOOL;
    A0XC0401_2_O_12 : BOOL;
    A0XC0401_2_O_13 : BOOL;
    A0XC0401_2_O_14 : BOOL;
    A0XC0401_2_O_15 : BOOL;
END_VAR
VAR_GLOBAL CONSTANT
    SC1501Ax : _sAXIS_REF;  (* at MC://_MC_AX[0] *)
    SC2301Ax : _sAXIS_REF;  (* at MC://_MC_AX[1] *)
    SC2302Ax : _sAXIS_REF;  (* at MC://_MC_AX[2] *)
    SC2303Ax : _sAXIS_REF;  (* at MC://_MC_AX[3] *)
    SC6401Ax : _sAXIS_REF;  (* at MC://_MC_AX[4] *)
END_VAR
VAR_GLOBAL
    XC0320_2_O_8 : BOOL;  (* at ECAT://node#10/Port2 Output Data01/Port2 Port5 Pin4 Output Bit *)
    XC0320_2_O_9 : BOOL;  (* at ECAT://node#10/Port2 Output Data01/Port2 Port5 Pin2 Output Bit *)
    fhfgn : BOOL;
    Module2_OUT_POW : BOOL;  (* at ECAT://node#10/Digital Output Data/Port2 Pin2 Digital Output Bit *)
    XC0320_1_I_2 : BOOL;
    XC0320_2_I_6 : BOOL;  (* Remote I/O Link Rotary Roller; at ECAT://node#10/Port2 Input Data01/Port2 Port4 Pin4 Input Bit *)
    XC0320_2_I_5 : BOOL;  (* Remote I/O Link Rotary Roller; at ECAT://node#10/Port2 Input Data01/Port2 Port3 Pin2 Input Bit *)
    XC0320_2_I_4 : BOOL;  (* Remote I/O Link Rotary Roller; at ECAT://node#10/Port2 Input Data01/Port2 Port3 Pin4 Input Bit *)
    XC0320_2_I_3 : BOOL;  (* Remote I/O Link Rotary Roller; at ECAT://node#10/Port2 Input Data01/Port2 Port2 Pin2 Input Bit *)
    XC0320_2_I_2 : BOOL;  (* Remote I/O Link Rotary Roller; at ECAT://node#10/Port2 Input Data01/Port2 Port2 Pin4 Input Bit *)
    XC0320_2_I_1 : BOOL;  (* Remote I/O Link Rotary Roller; at ECAT://node#10/Port2 Input Data01/Port2 Port1 Pin2 Input Bit *)
    XC0320_2_I_0 : BOOL;  (* Remote I/O Link Rotary Roller; at ECAT://node#10/Port2 Input Data01/Port2 Port1 Pin4 Input Bit *)
END_VAR

(* Program Program0: safety or other program stored in binary form, left out *)

PROGRAM Inputs
VAR
    DI3501_FB : MiscIN;
    DI3502_FB : MiscIN;
    PE3101_FB : MiscIN;
    PE3102_FB : MiscIN;
    PS2701_FB : MiscIN;
    PB0301_FB : MiscIN;
    PB0302_FB : MiscIN;
    PB0303_FB : MiscIN;
    SW0301_FB : MiscIN;
    PS0401_FB : MiscIN;
    PE1411_FB : MiscIN;
    PE1501_FB : MiscIN;
    PE1511_FB : MiscIN;
    PE1701_FB : MiscIN;
    PE1702_FB : MiscIN;
    PE1703_FB : MiscIN;
    PE1704_FB : MiscIN;
    PE1705_FB : MiscIN;
    PE1706_FB : MiscIN;
    PE1707_FB : MiscIN;
    PE1708_FB : MiscIN;
    PE2301_FB : MiscIN;
    PE2302FB : MiscIN;
    PE2303_FB : MiscIN;
    PE2304_FB : MiscIN;
    PE2305_FB : MiscIN;
    PE2701_FB : MiscIN;
    PE2702_FB : MiscIN;
    PE3601_FB : MiscIN;
    PE3602_FB : MiscIN;
    PE4101_FB : MiscIN;
    PE4102_FB : MiscIN;
    PE4103_FB : MiscIN;
    PE4111_FB : MiscIN;
    PE4112_FB : MiscIN;
    PE4113_FB : MiscIN;
    PE4114_FB : MiscIN;
    PE4121_FB : MiscIN;
    PE4122_FB : MiscIN;
    PE4123_FB : MiscIN;
    PE4124_FB : MiscIN;
    PS4101_FB : MiscIN;
    PS4102_FB : MiscIN;
    PS4103_FB : MiscIN;
    PS4104_FB : MiscIN;
    PS4111_FB : MiscIN;
    PS4112_FB : MiscIN;
    PS4113_FB : MiscIN;
    PS4114_FB : MiscIN;
    PS4121_FB : MiscIN;
    PS4122_FB : MiscIN;
    PS4123_FB : MiscIN;
    PS4124_FB : MiscIN;
    XC0303_EC_FB : MiscIN;
    MO3101_EC_FB : MiscIN;
    PE4104_FB : MiscIN;
    _EC : BOOL;
    XC0302_EC_FB : MiscIN;
    SC_EC_FB : MiscIN;
    SC3202_EC_FB : MiscIN;
    SC3201_EC_FB : MiscIN;
    SC3601_EC_FB : MiscIN;
    SC2701_EC_FB : MiscIN;
    SC1701_EC_FB : MiscIN;
    SC1702_EC_FB : MiscIN;
    MO2301_EC_FB : MiscIN;
    RO4001_EC_FB : MiscIN;
    RO4002_EC_FB : MiscIN;
    RO4003_EC_FB : MiscIN;
    XC0401_EC_FB : MiscIN;
    XC0411_EC_FB : MiscIN;
    OP0302_Ping : BOOL;
    OP0302_EC_FB : MiscIN;
    PE1401_FB : MiscIN;
    PE1402_FB : MiscIN;
    PE1403_FB : MiscIN;
    PE1601_FB : MiscIN;
    PE2201_FB : MiscIN;
    PE2202_FB : MiscIN;
    PE2203_FB : MiscIN;
    PE2204_FB : MiscIN;
    PE2205_FB : MiscIN;
    PE2206_FB : MiscIN;
    PE2302_FB : MiscIN;
    PX2301_FB : MiscIN;
    PE2311_FB : MiscIN;
    PE2312_FB : MiscIN;
    PE2313_FB : MiscIN;
    PE2314_FB : MiscIN;
    PE2315_FB : MiscIN;
    PE2316_FB : MiscIN;
    PE2317_FB : MiscIN;
    PE2401_FB : MiscIN;
    PE3103_FB : MiscIN;
    PE3104_FB : MiscIN;
    PE3401_FB : MiscIN;
    PE3402_FB : MiscIN;
    PE6901_FB : MiscIN;
    PE6902_FB : MiscIN;
    DI3503_FB : MiscIN;
    PX3401_FB : MiscIN;
    PS2501_FB : MiscIN;
    PE2306_FB : MiscIN;
    PE2307_FB : MiscIN;
    PE2308_FB : MiscIN;
    PE2309_FB : MiscIN;
    PX3101_FB : MiscIN;
    DI3301_FB : MiscIN;
    DI3302_FB : MiscIN;
    DI3303_FB : MiscIN;
    c : DINT;
    RO4001_TCPSpeed : WORD;
    PE1602_FB : MiscIN;
    DI3511_FB : MiscIN;
    PE3501_FB : MiscIN;
    A0XC0401_I3_8 : BOOL;
    PE3511_FB : MiscIN;
    PE3511 : MiscInD;
    PE1404_FB : MiscIN;
    PE6401_FB : MiscIN;
    PE1801_FB : MiscIN;
    PE1811_FB : MiscIN;
    PE1812_FB : MiscIN;
    PE1813_FB : MiscIN;
    PE1814_FB : MiscIN;
    PE1815_FB : MiscIN;
    PE2501_FB : MiscIN;
    PE2502_FB : MiscIN;
    PE2503_FB : MiscIN;
    PE2801_FB : MiscIN;
    PE2511_FB : MiscIN;
    PE2521_FB : MiscIN;
    PE2703_FB : MiscIN;
    PE7101_FB : MiscIN;
    PE2512_FB : MiscIN;
    PE6911_FB : MiscIN;
    PE6912_FB : MiscIN;
    DI0350_FB : MiscIN;
    DI7501_FB : MiscIN;
    DI7502_FB : MiscIN;
    DI7503_FB : MiscIN;
    DI3512_FB : MiscIN;
    DI3513_FB : MiscIN;
    PS2502_FB : MiscIN;
    PE6903_FB : MiscIN;
    PE6904_FB : MiscIN;
    jbcuevyq : BOOL;
    PX1801_FB : MiscIN;
END_VAR
VAR_EXTERNAL
    PE1501 : MiscInD;
    PE2201 : MiscInD;
    PE2202 : MiscInD;
    PE2203 : MiscInD;
    PE2301 : MiscInD;
    PE2302 : MiscInD;
    PE2303 : MiscInD;
    PE2401 : MiscInD;
    PE3401 : MiscInD;
    PE3402 : MiscInD;
    PE6901 : MiscInD;
    PE6902 : MiscInD;
    DI3511 : MiscInD;
    DI3501 : MiscInD;
    DI3502 : MiscInD;
    DI3503 : MiscInD;
    PS2501 : MiscInD;
    PS0401 : MiscInD;
    CY2502 : CylinderD;
    P27 : SequenceD;
    SV2501 : MiscOutD;
    RO4001_I_PalletizingDone : BOOL;
END_VAR
VAR_EXTERNAL CONSTANT
    _EC_CommErrTbl : ARRAY[1..256] OF BOOL;
    _EIP1_TDLinkAllRunSta : BOOL;
END_VAR
VAR_EXTERNAL
    PE1602 : MiscInD;
    PE3501 : MiscInD;
    PE1403 : MiscInD;
    PE1402 : MiscInD;
    PE1404 : MiscInD;
    PE6401 : MiscInD;
    PE1801 : MiscInD;
    PE1811 : MiscInD;
    PE1812 : MiscInD;
    PE1701 : MiscInD;
    PE1702 : MiscInD;
    PE2501 : MiscInD;
    PE2502 : MiscInD;
    PE2503 : MiscInD;
    PE2801 : MiscInD;
    PE2511 : MiscInD;
    PE2521 : MiscInD;
    PE2702 : MiscInD;
    PE2703 : MiscInD;
    PE7101 : MiscInD;
    PE3101 : MiscInD;
    PE2512 : MiscInD;
    PE6911 : MiscInD;
    PE6912 : MiscInD;
    DI0350 : MiscInD;
    DI7501 : MiscInD;
    DI7502 : MiscInD;
    DI7503 : MiscInD;
    DI3512 : MiscInD;
    DI3513 : MiscInD;
    XC0301_6_I : ARRAY[0..15] OF BOOL;
    PS2502 : MiscInD;
    XC0301_7_I : ARRAY[0..15] OF BOOL;
    XC0320_1_I_0 : BOOL;
    XC0320_1_I_1 : BOOL;
    XC0320_1_I_11 : BOOL;
    XC0320_1_I_12 : BOOL;
    XC0320_1_I_13 : BOOL;
    XC0320_1_I_14 : BOOL;
    XC0320_2_I_7 : BOOL;
    XC0320_2_I_8 : BOOL;
    XC0320_2_I_9 : BOOL;
    XC0320_2_I_10 : BOOL;
    XC0320_2_I_11 : BOOL;
    XC0320_2_I_12 : BOOL;
    XC0320_2_I_13 : BOOL;
    XC0320_2_I_14 : BOOL;
    XC0320_3_I_10 : BOOL;
    XC0320_3_I_11 : BOOL;
    PE6903 : MiscInD;
    PE6904 : MiscInD;
    XC0320_3_I_12 : BOOL;
    XC0320_3_I_13 : BOOL;
    XC0320_5_I_4 : BOOL;
    XC0320_5_I_5 : BOOL;
    XC0320_5_I_6 : BOOL;
    XC0320_5_I_7 : BOOL;
    A1_Control : System;
    PE1401 : MiscInD;
    XC0320_5_O_8 : BOOL;
    XC0320_5_O_9 : BOOL;
    XC0320_5_O_10 : BOOL;
    PE2701 : MiscInD;
    PE2204 : MiscInD;
    PE1703 : MiscInD;
    PE2206 : MiscInD;
    PE2205 : MiscInD;
    XC0320_1_I_15 : BOOL;
    XC0320_2_I_15 : BOOL;
    XC0320_3_I_6 : BOOL;
    XC0320_3_I_7 : BOOL;
    XC0320_3_I_8 : BOOL;
    XC0320_3_I_9 : BOOL;
    XC0320_4_I_8 : BOOL;
    XC0320_4_I_9 : BOOL;
    XC0320_4_I_10 : BOOL;
    XC0320_4_I_11 : BOOL;
    XC0320_4_I_12 : BOOL;
    XC0320_4_I_13 : BOOL;
    XC0320_4_I_14 : BOOL;
    XC0320_5_I_2 : BOOL;
    XC0320_5_I_3 : BOOL;
    PX1801 : MiscInD;
    XC0320_5_I_11 : BOOL;
    A0XC0401_1_I_0 : BOOL;
    A0XC0401_1_I_1 : BOOL;
    A0XC0401_1_I_3 : BOOL;
    A0XC0401_1_I_8 : BOOL;
    A0XC0401_1_I_9 : BOOL;
    A0XC0401_1_I_10 : BOOL;
    XC0320_4_I_15 : BOOL;
    XC0320_2_I_5 : BOOL;
    XC0320_2_I_6 : BOOL;
END_VAR

(* Section MiscInput: ladder, written here as Structured Text *)

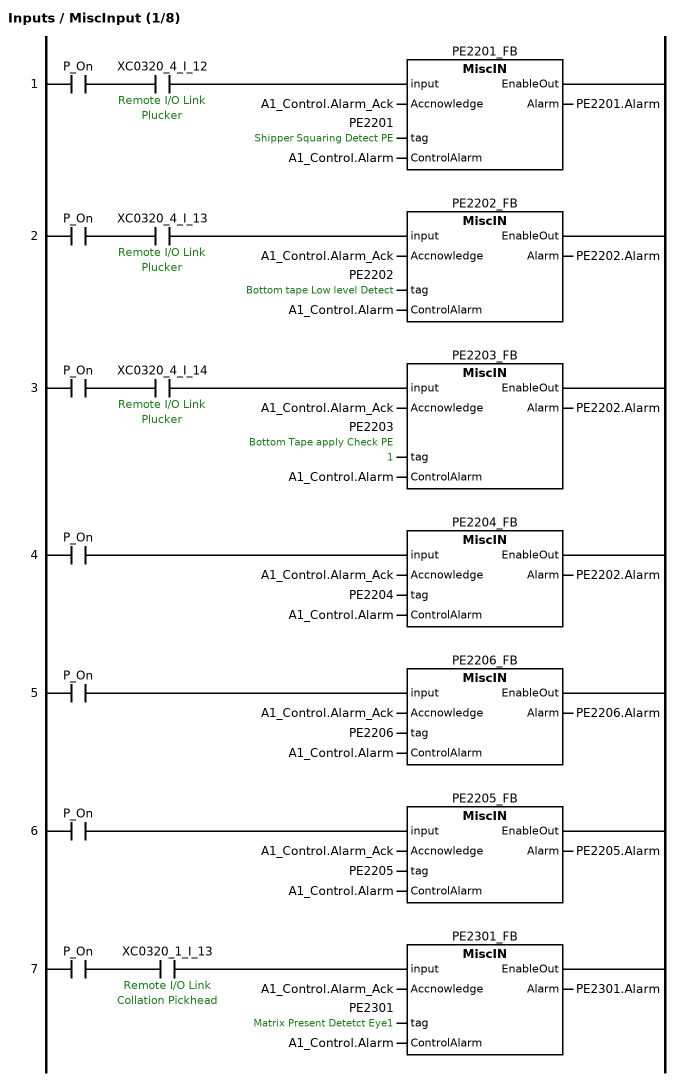
(* Rung 1 *)
PE2201_FB(input := P_On AND XC0320_4_I_12, Accnowledge := A1_Control.Alarm_Ack, tag := PE2201, ControlAlarm := A1_Control.Alarm, Alarm => PE2201.Alarm);
(* notes on elements: Pallet Presence Eye 1; Bottom Tapping Shipper Forming Detect PE *)
(* Rung 2 *)
PE2202_FB(input := P_On AND XC0320_4_I_13, Accnowledge := A1_Control.Alarm_Ack, tag := PE2202, ControlAlarm := A1_Control.Alarm, Alarm => PE2202.Alarm);
(* notes on elements: Bottom tape Low level Detect *)
(* Rung 3 *)
PE2203_FB(input := P_On AND XC0320_4_I_14, Accnowledge := A1_Control.Alarm_Ack, tag := PE2203, ControlAlarm := A1_Control.Alarm, Alarm => PE2202.Alarm);
(* notes on elements: Bottom Tape apply Check PE 1 *)
(* Rung 4 *)
PE2204_FB(input := P_On, Accnowledge := A1_Control.Alarm_Ack, tag := PE2204, ControlAlarm := A1_Control.Alarm, Alarm => PE2202.Alarm);
(* notes on elements: Bottom Tape apply Check PE 2 *)
(* Rung 5 *)
PE2206_FB(input := P_On, Accnowledge := A1_Control.Alarm_Ack, tag := PE2206, ControlAlarm := A1_Control.Alarm, Alarm => PE2206.Alarm);
(* notes on elements: Bottom Tape apply Check PE 2 *)
(* Rung 6 *)
PE2205_FB(input := P_On, Accnowledge := A1_Control.Alarm_Ack, tag := PE2205, ControlAlarm := A1_Control.Alarm, Alarm => PE2205.Alarm);
(* notes on elements: Bottom Tape apply Check PE 2 *)
(* Rung 7 *)
PE2301_FB(input := P_On AND XC0320_1_I_13, Accnowledge := A1_Control.Alarm_Ack, tag := PE2301, ControlAlarm := A1_Control.Alarm, Alarm => PE2301.Alarm);

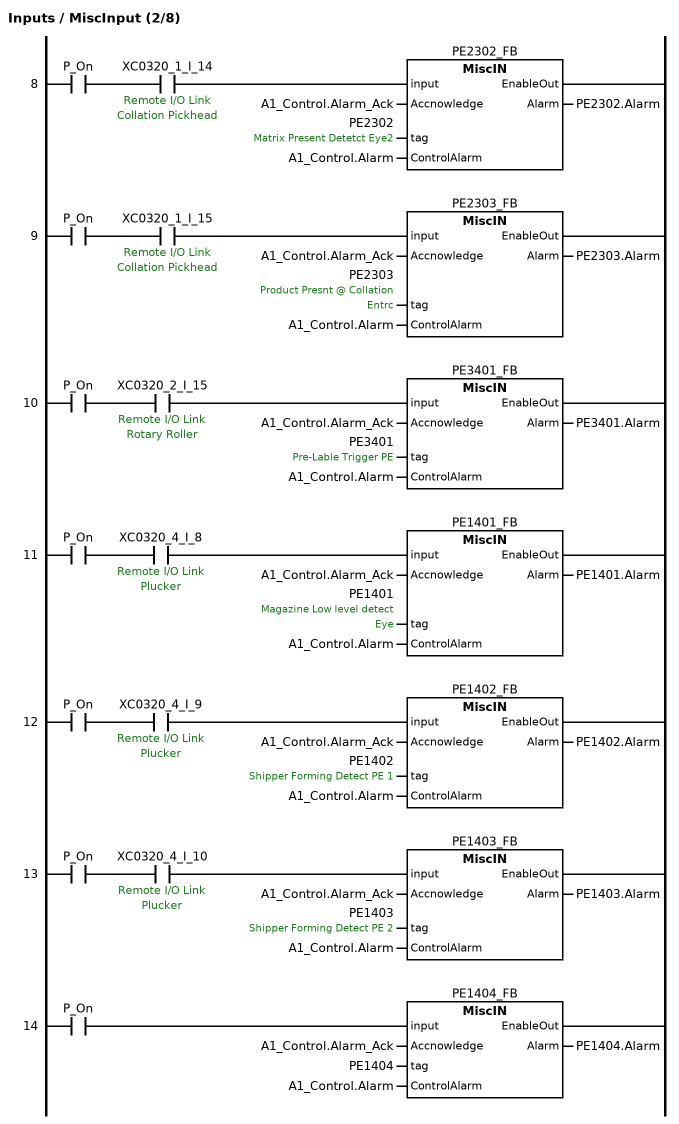
(* Rung 8 *)
PE2302_FB(input := P_On AND XC0320_1_I_14, Accnowledge := A1_Control.Alarm_Ack, tag := PE2302, ControlAlarm := A1_Control.Alarm, Alarm => PE2302.Alarm);
(* Rung 9 *)
PE2303_FB(input := P_On AND XC0320_1_I_15, Accnowledge := A1_Control.Alarm_Ack, tag := PE2303, ControlAlarm := A1_Control.Alarm, Alarm => PE2303.Alarm);
(* Rung 10 *)
PE3401_FB(input := P_On AND XC0320_2_I_15, Accnowledge := A1_Control.Alarm_Ack, tag := PE3401, ControlAlarm := A1_Control.Alarm, Alarm => PE3401.Alarm);
(* Rung 11 *)
PE1401_FB(input := P_On AND XC0320_4_I_8, Accnowledge := A1_Control.Alarm_Ack, tag := PE1401, ControlAlarm := A1_Control.Alarm, Alarm => PE1401.Alarm);
(* notes on elements: Magazine Low level detect Eye *)
(* Rung 12 *)
PE1402_FB(input := P_On AND XC0320_4_I_9, Accnowledge := A1_Control.Alarm_Ack, tag := PE1402, ControlAlarm := A1_Control.Alarm, Alarm => PE1402.Alarm);
(* notes on elements: Shipper Forming detect PE 1 *)
(* Rung 13 *)
PE1403_FB(input := P_On AND XC0320_4_I_10, Accnowledge := A1_Control.Alarm_Ack, tag := PE1403, ControlAlarm := A1_Control.Alarm, Alarm => PE1403.Alarm);
(* notes on elements: Shipper Forming detect PE 2 *)
(* Rung 14 *)
PE1404_FB(input := P_On, Accnowledge := A1_Control.Alarm_Ack, tag := PE1404, ControlAlarm := A1_Control.Alarm, Alarm => PE1404.Alarm);
(* notes on elements: Empty Level Detect PE *)

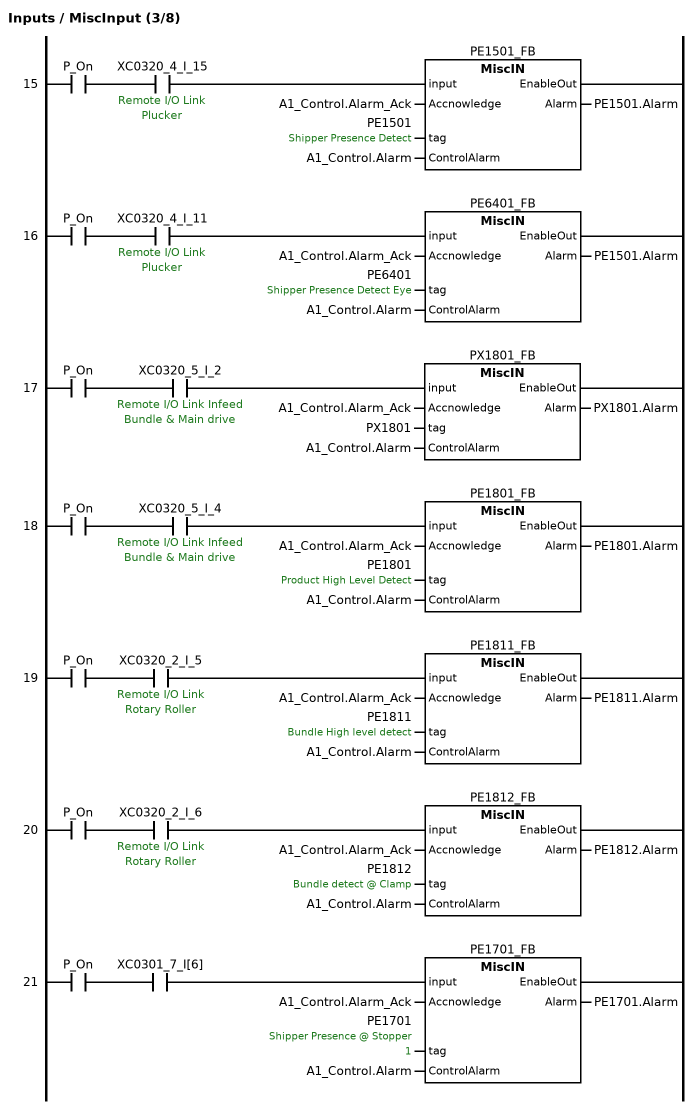
(* Rung 15 *)
PE1501_FB(input := P_On AND XC0320_4_I_15, Accnowledge := A1_Control.Alarm_Ack, tag := PE1501, ControlAlarm := A1_Control.Alarm, Alarm => PE1501.Alarm);
(* notes on elements: Shipper Presence Detect *)
(* Rung 16 *)
PE6401_FB(input := P_On AND XC0320_4_I_11, Accnowledge := A1_Control.Alarm_Ack, tag := PE6401, ControlAlarm := A1_Control.Alarm, Alarm => PE1501.Alarm);
(* notes on elements: Shipper Presence Detect *)
(* Rung 17 *)
PX1801_FB(input := P_On AND XC0320_5_I_2, Accnowledge := A1_Control.Alarm_Ack, tag := PX1801, ControlAlarm := A1_Control.Alarm, Alarm => PX1801.Alarm);
(* notes on elements: Conveyor lift detect Proxy *)
(* Rung 18 *)
PE1801_FB(input := P_On AND XC0320_5_I_4, Accnowledge := A1_Control.Alarm_Ack, tag := PE1801, ControlAlarm := A1_Control.Alarm, Alarm => PE1801.Alarm);
(* notes on elements: Product High Level Detect *)
(* Rung 19 *)
PE1811_FB(input := P_On AND XC0320_2_I_5, Accnowledge := A1_Control.Alarm_Ack, tag := PE1811, ControlAlarm := A1_Control.Alarm, Alarm => PE1811.Alarm);
(* notes on elements: Bundle High level detect *)
(* Rung 20 *)
PE1812_FB(input := P_On AND XC0320_2_I_6, Accnowledge := A1_Control.Alarm_Ack, tag := PE1812, ControlAlarm := A1_Control.Alarm, Alarm => PE1812.Alarm);
(* notes on elements: Product Detect @ clamp *)
(* Rung 21 *)
PE1701_FB(input := P_On AND XC0301_7_I[6], Accnowledge := A1_Control.Alarm_Ack, tag := PE1701, ControlAlarm := A1_Control.Alarm, Alarm => PE1701.Alarm);
(* notes on elements: Shipper Presence @ Stopper 1 *)

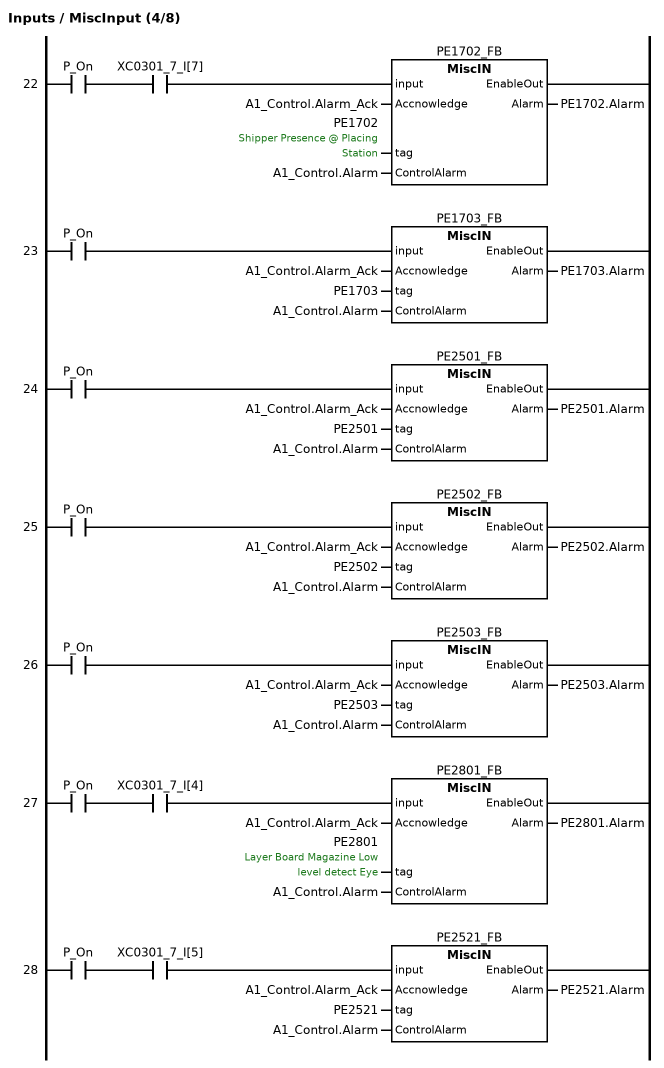
(* Rung 22 *)
PE1702_FB(input := P_On AND XC0301_7_I[7], Accnowledge := A1_Control.Alarm_Ack, tag := PE1702, ControlAlarm := A1_Control.Alarm, Alarm => PE1702.Alarm);
(* notes on elements: Shipper Presence @ Placing Station *)
(* Rung 23 *)
PE1703_FB(input := P_On, Accnowledge := A1_Control.Alarm_Ack, tag := PE1703, ControlAlarm := A1_Control.Alarm, Alarm => PE1703.Alarm);
(* notes on elements: Shipper Presence *)
(* Rung 24 *)
PE2501_FB(input := P_On, Accnowledge := A1_Control.Alarm_Ack, tag := PE2501, ControlAlarm := A1_Control.Alarm, Alarm => PE2501.Alarm);
(* notes on elements: Shipper Presence Detect Eye *)
(* Rung 25 *)
PE2502_FB(input := P_On, Accnowledge := A1_Control.Alarm_Ack, tag := PE2502, ControlAlarm := A1_Control.Alarm, Alarm => PE2502.Alarm);
(* notes on elements: Pickhead detect 1 @ changeover stand *)
(* Rung 26 *)
PE2503_FB(input := P_On, Accnowledge := A1_Control.Alarm_Ack, tag := PE2503, ControlAlarm := A1_Control.Alarm, Alarm => PE2503.Alarm);
(* notes on elements: Pickhead detect 2 @ changeover stand *)
(* Rung 27 *)
PE2801_FB(input := P_On AND XC0301_7_I[4], Accnowledge := A1_Control.Alarm_Ack, tag := PE2801, ControlAlarm := A1_Control.Alarm, Alarm => PE2801.Alarm);
(* notes on elements: Layer Board Magazine Low level detect Eye *)
(* Rung 28 *)
PE2521_FB(input := P_On AND XC0301_7_I[5], Accnowledge := A1_Control.Alarm_Ack, tag := PE2521, ControlAlarm := A1_Control.Alarm, Alarm => PE2521.Alarm);
(* notes on elements: Product Presence *)

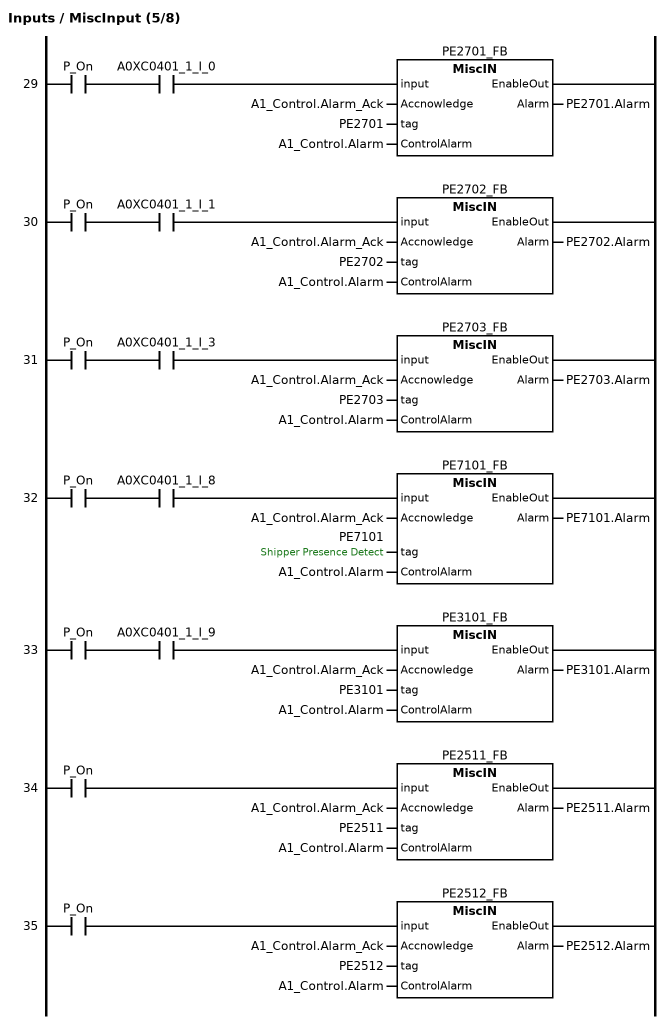
(* Rung 29 *)
PE2701_FB(input := P_On AND A0XC0401_1_I_0, Accnowledge := A1_Control.Alarm_Ack, tag := PE2701, ControlAlarm := A1_Control.Alarm, Alarm => PE2701.Alarm);
(* notes on elements: Box Present detect PE1 *)
(* Rung 30 *)
PE2702_FB(input := P_On AND A0XC0401_1_I_1, Accnowledge := A1_Control.Alarm_Ack, tag := PE2702, ControlAlarm := A1_Control.Alarm, Alarm => PE2702.Alarm);
(* notes on elements: Box detect PE2 *)
(* Rung 31 *)
PE2703_FB(input := P_On AND A0XC0401_1_I_3, Accnowledge := A1_Control.Alarm_Ack, tag := PE2703, ControlAlarm := A1_Control.Alarm, Alarm => PE2703.Alarm);
(* notes on elements: Top Tapping Low level *)
(* Rung 32 *)
PE7101_FB(input := P_On AND A0XC0401_1_I_8, Accnowledge := A1_Control.Alarm_Ack, tag := PE7101, ControlAlarm := A1_Control.Alarm, Alarm => PE7101.Alarm);
(* notes on elements: Shipper Presence Detect *)
(* Rung 33 *)
PE3101_FB(input := P_On AND A0XC0401_1_I_9, Accnowledge := A1_Control.Alarm_Ack, tag := PE3101, ControlAlarm := A1_Control.Alarm, Alarm => PE3101.Alarm);
(* notes on elements: Shipper Presence Detect *)
(* Rung 34 *)
PE2511_FB(input := P_On, Accnowledge := A1_Control.Alarm_Ack, tag := PE2511, ControlAlarm := A1_Control.Alarm, Alarm => PE2511.Alarm);
(* notes on elements: Shipper Presence Detect Eye 1 *)
(* Rung 35 *)
PE2512_FB(input := P_On, Accnowledge := A1_Control.Alarm_Ack, tag := PE2512, ControlAlarm := A1_Control.Alarm, Alarm => PE2512.Alarm);
(* notes on elements: Shipper Presence Detect Eye 2 *)

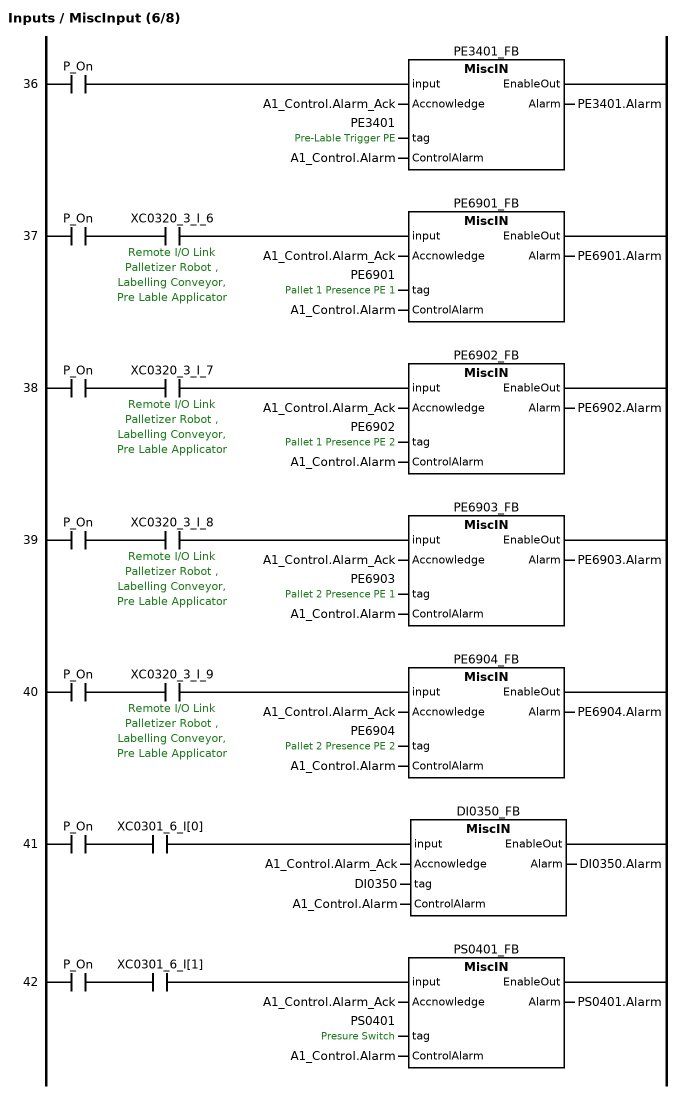
(* Rung 36 *)
PE3401_FB(input := P_On, Accnowledge := A1_Control.Alarm_Ack, tag := PE3401, ControlAlarm := A1_Control.Alarm, Alarm => PE3401.Alarm);
(* notes on elements: Shipper Presence Detect Eye *)
(* Rung 37 *)
PE6901_FB(input := P_On AND XC0320_3_I_6, Accnowledge := A1_Control.Alarm_Ack, tag := PE6901, ControlAlarm := A1_Control.Alarm, Alarm => PE6901.Alarm);
(* notes on elements: Pallet Presence Eye 1 *)
(* Rung 38 *)
PE6902_FB(input := P_On AND XC0320_3_I_7, Accnowledge := A1_Control.Alarm_Ack, tag := PE6902, ControlAlarm := A1_Control.Alarm, Alarm => PE6902.Alarm);
(* notes on elements: Pallet Presence Eye 2 *)
(* Rung 39 *)
PE6903_FB(input := P_On AND XC0320_3_I_8, Accnowledge := A1_Control.Alarm_Ack, tag := PE6903, ControlAlarm := A1_Control.Alarm, Alarm => PE6903.Alarm);
(* notes on elements: Pallet 2 Presence Eye 1 *)
(* Rung 40 *)
PE6904_FB(input := P_On AND XC0320_3_I_9, Accnowledge := A1_Control.Alarm_Ack, tag := PE6904, ControlAlarm := A1_Control.Alarm, Alarm => PE6904.Alarm);
(* notes on elements: Pallet 2 Presence Eye 1 *)
(* Rung 41 *)
DI0350_FB(input := P_On AND XC0301_6_I[0], Accnowledge := A1_Control.Alarm_Ack, tag := DI0350, ControlAlarm := A1_Control.Alarm, Alarm => DI0350.Alarm);
(* notes on elements: Rejection Table Full PE 2 *)
(* Rung 42 *)
PS0401_FB(input := P_On AND XC0301_6_I[1], Accnowledge := A1_Control.Alarm_Ack, tag := PS0401, ControlAlarm := A1_Control.Alarm, Alarm => PS0401.Alarm);
(* notes on elements: Presure Switch *)

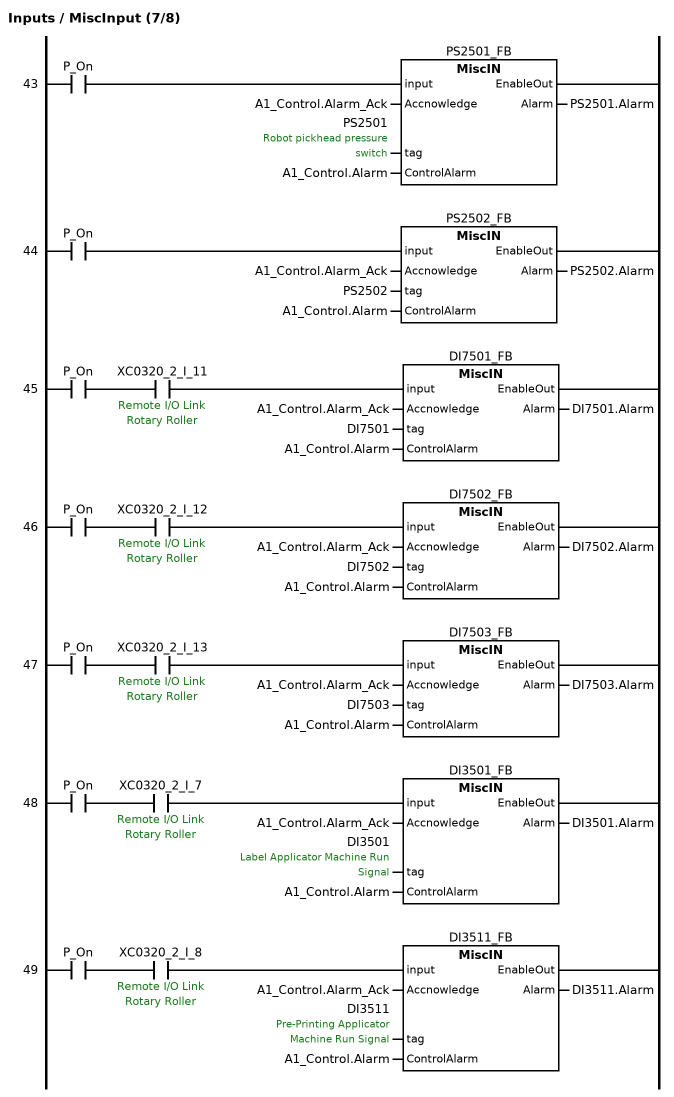
(* Rung 43 *)
PS2501_FB(input := P_On, Accnowledge := A1_Control.Alarm_Ack, tag := PS2501, ControlAlarm := A1_Control.Alarm, Alarm => PS2501.Alarm);
(* notes on elements: Pressure Switch 1 *)
(* Rung 44 *)
PS2502_FB(input := P_On, Accnowledge := A1_Control.Alarm_Ack, tag := PS2502, ControlAlarm := A1_Control.Alarm, Alarm => PS2502.Alarm);
(* notes on elements: Pressure Switch 2 *)
(* Rung 45 *)
DI7501_FB(input := P_On AND XC0320_2_I_11, Accnowledge := A1_Control.Alarm_Ack, tag := DI7501, ControlAlarm := A1_Control.Alarm, Alarm => DI7501.Alarm);
(* notes on elements: Checkweigher Run Signal *)
(* Rung 46 *)
DI7502_FB(input := P_On AND XC0320_2_I_12, Accnowledge := A1_Control.Alarm_Ack, tag := DI7502, ControlAlarm := A1_Control.Alarm, Alarm => DI7502.Alarm);
(* notes on elements: Checkweigher Accept Signal *)
(* Rung 47 *)
DI7503_FB(input := P_On AND XC0320_2_I_13, Accnowledge := A1_Control.Alarm_Ack, tag := DI7503, ControlAlarm := A1_Control.Alarm, Alarm => DI7503.Alarm);
(* notes on elements: Checkweigher Reject Signal *)
(* Rung 48 *)
DI3501_FB(input := P_On AND XC0320_2_I_7, Accnowledge := A1_Control.Alarm_Ack, tag := DI3501, ControlAlarm := A1_Control.Alarm, Alarm => DI3501.Alarm);
(* notes on elements: Pre-Label Applicator Machine Run Signal *)
(* Rung 49 *)
DI3511_FB(input := P_On AND XC0320_2_I_8, Accnowledge := A1_Control.Alarm_Ack, tag := DI3511, ControlAlarm := A1_Control.Alarm, Alarm => DI3511.Alarm);
(* notes on elements: OCR Camera Run Signal *)

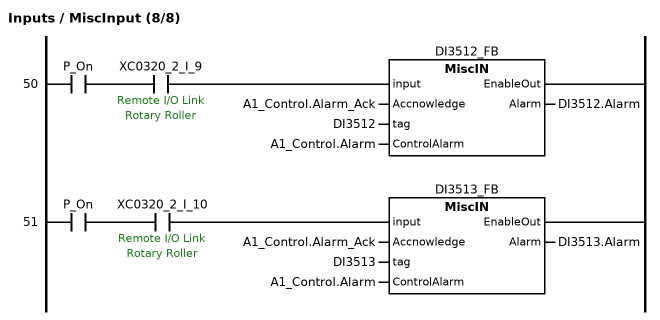
(* Rung 50 *)
DI3512_FB(input := P_On AND XC0320_2_I_9, Accnowledge := A1_Control.Alarm_Ack, tag := DI3512, ControlAlarm := A1_Control.Alarm, Alarm => DI3512.Alarm);
(* notes on elements: OCR Camera Accept Signal *)
(* Rung 51 *)
DI3513_FB(input := P_On AND XC0320_2_I_10, Accnowledge := A1_Control.Alarm_Ack, tag := DI3513, ControlAlarm := A1_Control.Alarm, Alarm => DI3513.Alarm);
(* notes on elements: OCR Camera Reject Signal *)

(* Section IDRob_Inputs: ladder, written here as Structured Text *)

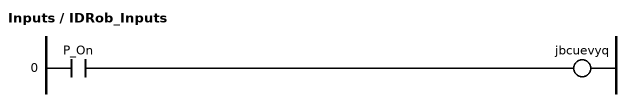
(* Rung 0 *)
jbcuevyq := P_On;

(* Section IDRob_SysInputs: ladder, written here as Structured Text *)

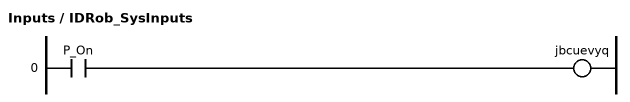
(* Rung 0 *)
jbcuevyq := P_On;
END_PROGRAM

PROGRAM Control
VAR
    EmergencyStopOK : BOOL;
    GuardDoorsOK : BOOL;
    ClearingTime : TIME;
    ClearingTimer : TON;
    BlinkTimer1 : TON;
    Blink : BOOL;
    BlinkTimer2 : TON;
    Reset_Timer : BOOL;
    Reset_Timer1 : BOOL;
    Statistics_Timer : TON;
    Stat_time : TIME;
    Time1 : TIME;
    CartonsPerMin1 : ARRAY[0..2] OF LREAL;
    Cycle_Time : TIME;
    Temp : TIME;
    Total_RunHours1 : TIME;
    Cycle_TIme_NanoSec : LINT;
    Cycle_TIme_NanoSec1 : LREAL;
    Cycle_Time_Microsec : LREAL;
    Cycle_Time_Milisec : LREAL;
    Total_RunHours2 : TIME;
    Total_RunHours3 : LINT;
    Total_RunHours4 : LINT;
    Total_RunHours5 : LREAL;
    Total_RunHours : TON;
    P14_StepEngine : Stepengine;
    P15_StepEngine : StepEngine;
    P31_StepEngine : StepEngine;
    P27_StepEngine : StepEngine;
    P18_StepEngine : StepEngine;
    P17_StepEngine : StepEngine;
    P18b_StepEngine : StepEngine;
    P31a_StepEngine : StepEngine;
    P31b_StepEngine : StepEngine;
    P15b_StepEngine : StepEngine;
    P15a_StepEngine : StepEngine;
    P18a_StepEngine : StepEngine;
    P14a_StepEngine : StepEngine;
    P36_StepEngine : StepEngine;
    Tracking_ONS : ARRAY[0..9] OF BOOL;
    Track : DINT;
    P32_StepEngine : StepEngine;
    P15c_StepEngine : StepEngine;
    Executiontime : TIME;
    ExecutionTime1 : LINT;
    ExecutionTime2 : REAL;
    EthercatError_reset : ResetECError;
    PLCError_Reset : ResetPLCError;
    Reset_Runtimer : BOOL;
    Selected_Recipe : DINT;
    Completetimer : TON;
    P15d_StepEngine : StepEngine;
    Step_1 : TON;
    Step_2 : TON;
    Step_3 : TON;
    Step_4 : TON;
    CA1701_TMR_1 : TON;
    CA1701_TMR_2 : TON;
    CA1701_TMR_3 : TON;
    P24_StepEngine : StepEngine;
    P23b_StepEngine : StepEngine;
    P23a_StepEngine : StepEngine;
    P23_StepEngine : StepEngine;
    P22_StepEngine : StepEngine;
    P34_StepEngine : StepEngine;
    P40_StepEngine : StepEngine;
    P23c_StepEngine : StepEngine;
    MotionError_Reset : ResetMCError;
    P23d_StepEngine : StepEngine;
    uygwurgf : BOOL;
    kfbejwvb : BOOL;
    bcjwebjvb : BOOL;
    ckbed : BOOL;
    TrackShipper : TON;
    taping_timer1 : TON;
    Matrix_timing : TON;
    movetopos1manual : BOOL;
    RO4001_I_M : BOOL;
    RO4001Start : BOOL;
    RO4001Starttimer : TON;
    RO4001Motorontimer : TON;
    RO4001Motorontimer1 : TON;
    Carton_Per_Shipper : DINT;
    Carton_Per_box : DINT;
    No_of_Layers : REAL;
    RO4001_I_ShipperPickPermit : BOOL;
    RO4001_I_ShipperP : BOOL;
    RO4001_I_Matrix : BOOL;
    zcom : BOOL;
    PPMAinTImer : TON;
    IPCchecktimer : TON;
    IPCchecktimer1 : TON;
    IPCchecktimer2 : TON;
    IPCchecktimer3 : TON;
    P22_TopCount : DINT;
    TapeCheck : DINT;
    P22_BottomCount : DINT;
    BottomTapeLowCount : DINT;
    TopTapeLowCount : DINT;
    PE : BOOL;
    zcomm12 : BOOL;
    jbcuevyq : BOOL;
    P64_StepEngine : StepEngine;
    P28_StepEngine : StepEngine;
    P71_StepEngine : StepEngine;
    Collation_Unit_1_Rows : CTU;
    Collation_Unit_2_Rows : CTU;
    PartionCheck_Timer : TON;
    Write_data : IOL_WriteObj;
    Dport : INT;
    DevObj : _sIOLOBJ_ACCESS;
    WrtData : INT;
    err : BOOL;
    Test_Bit : BOOL;
    ErrID : WORD;
    ErrTyp : WORD;
    Dport1 : _sDEVICE_PORT;
    Zcom13 : BOOL;
    Zcom14 : BOOL;
    SC1501_Home : MC_Home;
    Home_Temp : BOOL;
    XC0301_6_I0 : BOOL;
END_VAR
VAR RETAIN
    SC2301_Temp1 : LREAL;  (* Side Shifting Position for Recipe POS1 *)
END_VAR
VAR
    Stopper_CYL_Pos_From_Infeed : LREAL;
    Infeed_Belt_Width : REAL;
    SC2301_Pos1_Fixed_target : LREAL;  (* SC2301_Pos1_Close_To_Infeed *)
END_VAR
VAR RETAIN
    SC2301_Temp2 : LREAL;  (* SC2301_Position_cal_At_Infeed *)
    SC2301_Temp3 : LREAL;  (* SC2301_Pos_For_Big_Product_Width *)
END_VAR
VAR
    Z : BOOL;
    Zcom20 : BOOL;
    sgdsfg : BOOL;
    P : BOOL;
    ZCOM29 : BOOL;
    DRY_CYCLE : BOOL;
    ZCOM34 : BOOL;
    zcom15 : BOOL;
    zcom16 : BOOL;
    zcom17 : BOOL;
    ZCOM18 : BOOL;
    ZCOM19 : BOOL;
    ZCOM21 : BOOL;
    SC2302_Temp1 : LREAL;
    SC2302_Temp2 : LREAL;
END_VAR
VAR RETAIN
    Robot_Pick_No_Collation_1 : LREAL;
END_VAR
VAR
    RO6301_I_Product_Pick_Count : LREAL;
    Produc_count_OK : INT;
    Count_Trig : R_TRIG;
    zcom22 : BOOL;
    zcom23 : BOOL;
    zcom24 : BOOL;
    Zcom25 : BOOL;
    SC2301_Temp4 : LREAL;
    zcom26 : BOOL;
    zcom27 : BOOL;
    dfbvv : BOOL;
    afadfv : BOOL;
    adfcascv : BOOL;
    acsavas : BOOL;
    sfgadfvad : BOOL;
    aefgaefgvedf : BOOL;
END_VAR
VAR RETAIN
    SC2303_Temp1 : LREAL;  (* SC2303_Fix_Position_Near_Infeed *)
    SC2303_Temp2 : LREAL;
    SC2303_Temp3 : LREAL;
    SC2303_Temp4 : LREAL;
END_VAR
VAR
    Zcommm : BOOL;
    Zzcom : BOOL;
    Zdfsdf : BOOL;
    dfgdfh : BOOL;
    vcvfb : BOOL;
    hffgdgn : BOOL;
    fgjghkg : BOOL;
    dsvdfdf : BOOL;
    dsgsfgdfgh : BOOL;
    sfgf : BOOL;
    Start_Timer : TON;
END_VAR
VAR_EXTERNAL
    A1_Control : System;
    MO1402 : MotorD;
    P23c : SequenceD;
    SafetyDeviceReady : BOOL;
    IL0301 : MiscOutD;
    IL0302 : MiscOutD;
    IL0303 : MiscOutD;
    Batch_Report : BatchDetails;
    SV1501 : MiscOutD;
    PE1501 : MiscInD;
    PE2203 : MiscInD;
    MO2201 : MotorD;
    MO2202 : MotorD;
    CY2301 : CylinderD;
    CY2401 : CylinderD;
    CY2402 : CylinderD;
    PE2401 : MiscInD;
    SC2701 : ServoD;
    CY1601 : CylinderD;
    PE3401 : MiscInD;
    Shipper_Accept : BOOL;
    CY2304 : CylinderD;
    Reject_Matrix_Accept : BOOL;
    Carton_Matrix_Accept : BOOL;
    CY2302 : CylinderD;
    CY2303 : CylinderD;
    RO4001_I_PalletizingDone : BOOL;
    Palletizing_Done : BOOL;
    PE6901 : MiscInD;
    PE6902 : MiscInD;
    PE2201 : MiscInD;
    PE2202 : MiscInD;
    DI3501 : MiscInD;
    DI3502 : MiscInD;
    Shipper_Reject : BOOL;
    Shipper_Good_Count : BOOL;
    S_CellEnabled : BOOL;
    PE2302 : MiscInD;
    SKU_Select : DINT;
    PE2301 : MiscInD;
    PE2303 : MiscInD;
    P27 : SequenceD;
    MO2301 : MotorD;
    SV2301 : MiscOutD;
    PE3402 : MiscInD;
    SV2501 : MiscOutD;
    SV2502 : MiscOutD;
    CY2501 : CylinderD;
    TotalLayers : DINT;
    ShippersPerLayer : DINT;
    IPCcheck : BOOL;
    IPCcheckAlarm : BOOL;
    IPCCheck1 : BOOL;
    P22_TapeAlarm : BOOL;
    PS2501 : MiscInD;
    RO4001_Alarm : BOOL;
    RO4001_ErrorTrigger : ARRAY[0..9] OF BOOL;
    PE3501 : MiscInD;
    DO3502 : MiscOutD;
    DO3501 : MiscOutD;
    K1301 : MiscOutD;
    SV2701 : MiscOutD;
    RESET_CMD : BOOL;
    ES1001_I : BOOL;
    ES1201_I : BOOL;
    ES4001_I : BOOL;
    GZ1301_I : BOOL;
    GZ1302_I : BOOL;
    P22 : SequenceD;
    abc : INT;
    efd : INT;
    dsg : LREAL;
    CH : INT;
    Recipe : RecipeD;
    SKU_No : DINT;
    ES1202_I : BOOL;
    ES1203_I : BOOL;
    GZ1303_I : BOOL;
    GZ1304_I : BOOL;
    GZ1305_I : BOOL;
    P15 : SequenceD;
    P64 : SequenceD;
    P14 : SequenceD;
    P18A : SequenceD;
    P23 : SequenceD;
    P17 : SequenceD;
    P18 : SequenceD;
    P28 : SequenceD;
    P71 : SequenceD;
    PE1401 : MiscInD;
    SC1501 : ServoD;
    CY1501 : CylinderD;
    CY1502 : CylinderD;
    CY1503 : CylinderD;
    CY1504 : CylinderD;
    PE6401 : MiscInD;
    SC6401 : ServoD;
    P23a : SequenceD;
    SC2301 : ServoD;
    SC2302 : ServoD;
    Collation_Unit_1_Define_RowsNo : REAL;
    Collation_Unit_1_Running_RowsNo : INT;
    Product_Width : REAL;
    SC2301_Pos2_Variable_1 : LREAL;
    SC2301_Pos2_Temp1 : REAL;
    SC2301_Pos2_Temp2 : REAL;
    SC2302_Pos2_Temp1 : REAL;
    SC2301_Pos3_Temp1 : REAL;
    RO6301_Flag : BOOL;
    PE1811 : MiscInD;
    SC2303 : ServoD;
    Collation_Unit_2_Define_RowsNo : REAL;
    SC2303_Pos2_Temp1 : REAL;
    SC2302_Pos4_Temp1 : REAL;
    Collation_Unit_1_Define_RowsNo_INT : INT;
    Collation_Unit_2_Define_RowsNo_INT : INT;
    PE1701 : MiscInD;
    CY1702 : CylinderD;
    CY1701 : CylinderD;
    PE1702 : MiscInD;
    CY1703 : CylinderD;
    RO6101_MatrixPlace : BOOL;
    RO6102_PartionPlace : BOOL;
    PE7101 : MiscInD;
    CY7101 : CylinderD;
    CY7102 : CylinderD;
    PE1402 : MiscInD;
    PE1403 : MiscInD;
    MO1801 : MotorD;
    PE2801 : MiscInD;
    PE2205 : MiscInD;
    ydytdutf : BOOL;
    ujcjgcj : BOOL;
    khvjk : BOOL;
    hkfvkhf : BOOL;
END_VAR
VAR_EXTERNAL CONSTANT
    SC1501Ax : _sAXIS_REF;
END_VAR
VAR_EXTERNAL
    Zcomm : ARRAY[0..31] OF BOOL;
    XC0301_6_I : ARRAY[0..15] OF BOOL;
    MO1401 : MotorD;
    SV1502 : MiscOutD;
    SV1503 : MiscOutD;
    fhfgn : BOOL;
    Module2_OUT_POW : BOOL;
    CY1811 : CylinderD;
    CY2305 : CylinderD;
    MO1811 : MotorD;
    MO1802 : MotorD;
    MO1701 : MotorD;
END_VAR
VAR
    _p1 : BOOL;
    _e2 : R_TRIG;
    _p3 : BOOL;
    _p4 : BOOL;
    _p5 : BOOL;
    _p6 : BOOL;
    _e7 : R_TRIG;
    _e8 : R_TRIG;
    _p9 : BOOL;
    _e10 : R_TRIG;
    _e11 : R_TRIG;
    _e12 : R_TRIG;
    _e13 : R_TRIG;
    _e14 : R_TRIG;
    _e15 : R_TRIG;
    _p16 : BOOL;
    _e17 : R_TRIG;
    _e18 : R_TRIG;
    _p19 : BOOL;
    _p20 : BOOL;
    _e21 : R_TRIG;
    _p22 : BOOL;
    _e23 : R_TRIG;
    _p24 : BOOL;
    _e25 : R_TRIG;
    _e26 : R_TRIG;
    _p27 : BOOL;
    _p28 : BOOL;
    _p29 : BOOL;
    _p30 : BOOL;
    _e31 : R_TRIG;
    _e32 : R_TRIG;
    _p33 : BOOL;
    _p34 : BOOL;
    _p35 : BOOL;
    _p36 : BOOL;
    _e37 : R_TRIG;
    _p38 : BOOL;
    _e39 : R_TRIG;
    _e40 : R_TRIG;
    _e41 : R_TRIG;
    _p42 : BOOL;
    _p43 : BOOL;
    _p44 : BOOL;
    _e45 : R_TRIG;
    _e46 : R_TRIG;
    _p47 : BOOL;
    _p48 : BOOL;
    _p49 : BOOL;
    _e50 : R_TRIG;
    _p51 : BOOL;
    _e52 : R_TRIG;
    _e53 : R_TRIG;
    _e54 : R_TRIG;
    _p55 : BOOL;
    _e56 : R_TRIG;
    _e57 : R_TRIG;
    _e58 : R_TRIG;
    _t59 : DINT;
    _e60 : R_TRIG;
    _e61 : R_TRIG;
    _e62 : R_TRIG;
    _p63 : BOOL;
    _e64 : R_TRIG;
    _e65 : R_TRIG;
END_VAR

(* Section Safety: ladder, written here as Structured Text *)

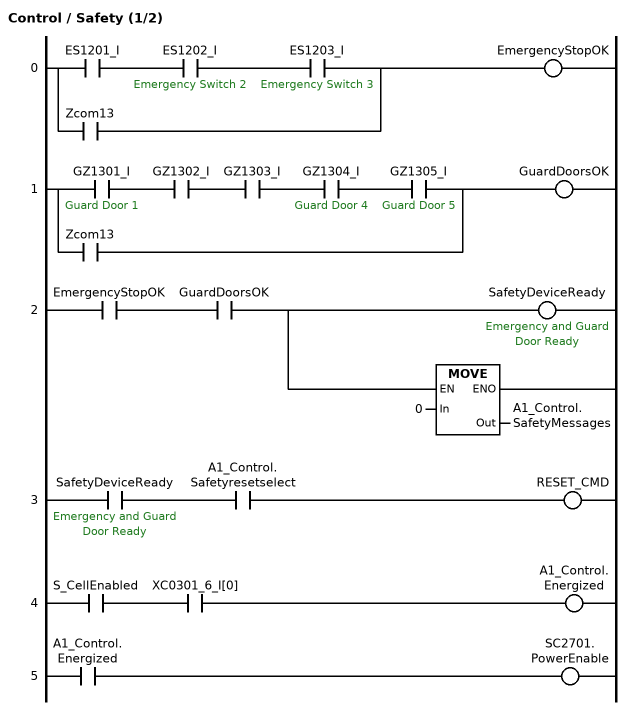
(* Rung 0 *)
EmergencyStopOK := (ES1201_I AND ES1202_I AND ES1203_I) OR Zcom13;
(* Rung 1 *)
GuardDoorsOK := (GZ1301_I AND GZ1302_I AND GZ1303_I AND GZ1304_I AND GZ1305_I) OR Zcom13;
(* Rung 2 *)
SafetyDeviceReady := EmergencyStopOK AND GuardDoorsOK;
IF EmergencyStopOK AND GuardDoorsOK THEN A1_Control.SafetyMessages := 0; END_IF;
(* Rung 3 *)
RESET_CMD := SafetyDeviceReady AND A1_Control.Safetyresetselect;
(* Rung 4 *)
A1_Control.Energized := S_CellEnabled AND XC0301_6_I[0];
(* Rung 5 *)
SC2701.PowerEnable := A1_Control.Energized;

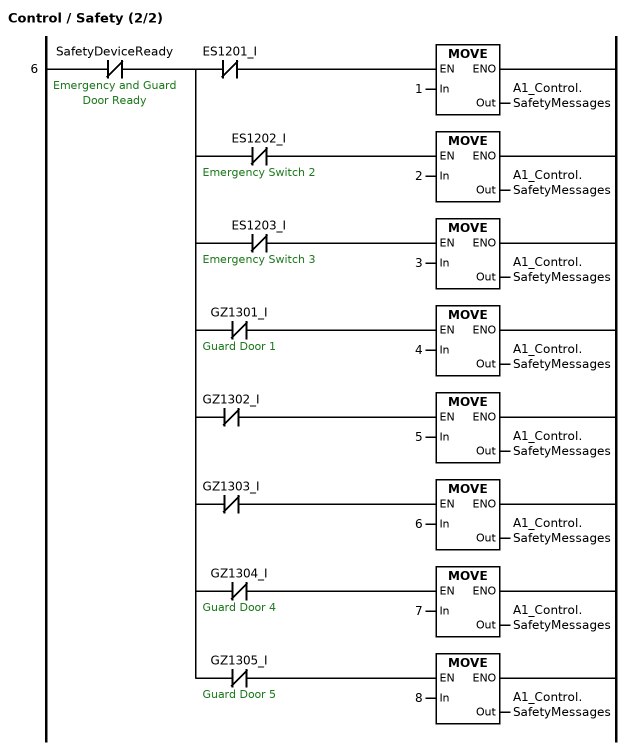
(* Rung 6 *)
IF NOT SafetyDeviceReady AND NOT ES1201_I THEN A1_Control.SafetyMessages := 1; END_IF;
IF NOT SafetyDeviceReady AND NOT ES1202_I THEN A1_Control.SafetyMessages := 2; END_IF;
IF NOT SafetyDeviceReady AND NOT ES1203_I THEN A1_Control.SafetyMessages := 3; END_IF;
IF NOT SafetyDeviceReady AND NOT GZ1301_I THEN A1_Control.SafetyMessages := 4; END_IF;
IF NOT SafetyDeviceReady AND NOT GZ1302_I THEN A1_Control.SafetyMessages := 5; END_IF;
IF NOT SafetyDeviceReady AND NOT GZ1303_I THEN A1_Control.SafetyMessages := 6; END_IF;
IF NOT SafetyDeviceReady AND NOT GZ1304_I THEN A1_Control.SafetyMessages := 7; END_IF;
IF NOT SafetyDeviceReady AND NOT GZ1305_I THEN A1_Control.SafetyMessages := 8; END_IF;

(* Section Control: ladder, written here as Structured Text *)

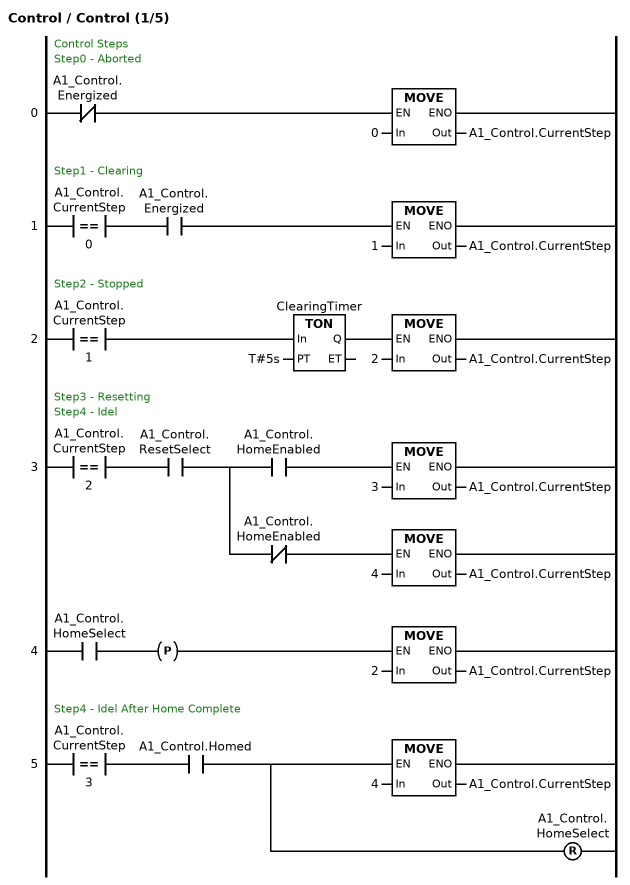
(* Rung 0: Control Steps / Step0 - Aborted *)
IF NOT A1_Control.Energized THEN A1_Control.CurrentStep := 0; END_IF;
(* Rung 1: Step1 - Clearing *)
IF (A1_Control.CurrentStep = 0) AND A1_Control.Energized THEN A1_Control.CurrentStep := 1; END_IF;
(* Rung 2: Step2 - Stopped *)
ClearingTimer(In := A1_Control.CurrentStep = 1, PT := T#5s);
IF ClearingTimer.Q THEN A1_Control.CurrentStep := 2; END_IF;
(* Rung 3: Step3 - Resetting / Step4 - Idel *)
_p1 := (A1_Control.CurrentStep = 2) AND A1_Control.ResetSelect;
IF _p1 AND A1_Control.HomeEnabled THEN A1_Control.CurrentStep := 3; END_IF;
IF _p1 AND NOT A1_Control.HomeEnabled THEN A1_Control.CurrentStep := 4; END_IF;
(* Rung 4 *)
_e2(CLK := A1_Control.HomeSelect);
IF _e2.Q THEN A1_Control.CurrentStep := 2; END_IF;
(* Rung 5: Step4 - Idel After Home Complete *)
_p3 := (A1_Control.CurrentStep = 3) AND A1_Control.Homed;
IF _p3 THEN
    A1_Control.CurrentStep := 4;
    A1_Control.HomeSelect := FALSE;
END_IF;

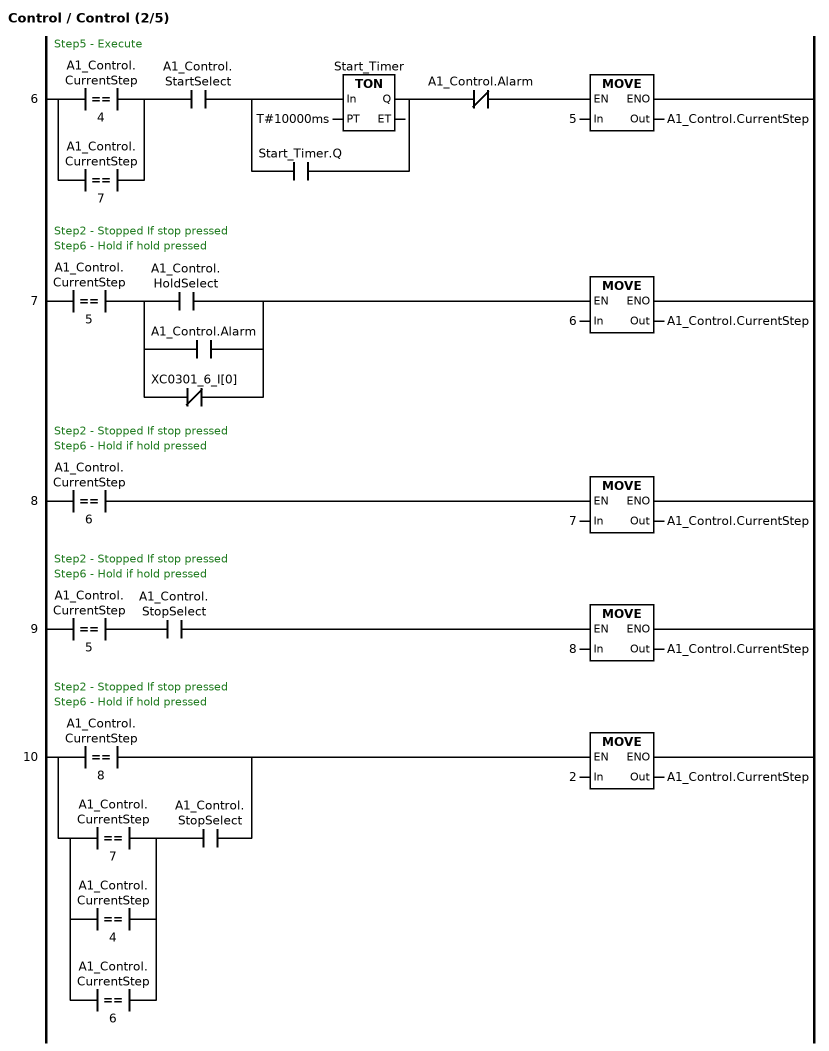
(* Rung 6: Step5 - Execute *)
_p4 := ((A1_Control.CurrentStep = 4) OR (A1_Control.CurrentStep = 7)) AND A1_Control.StartSelect;
Start_Timer(In := _p4, PT := T#10000ms);
IF (Start_Timer.Q OR (_p4 AND Start_Timer.Q)) AND NOT A1_Control.Alarm THEN
    A1_Control.CurrentStep := 5;
END_IF;
(* Rung 7: Step2 - Stopped If stop pressed / Step6 - Hold if hold pressed *)
IF (A1_Control.CurrentStep = 5) AND (A1_Control.HoldSelect OR A1_Control.Alarm OR NOT XC0301_6_I[0]) THEN
    A1_Control.CurrentStep := 6;
END_IF;
(* Rung 8: Step2 - Stopped If stop pressed / Step6 - Hold if hold pressed *)
IF A1_Control.CurrentStep = 6 THEN A1_Control.CurrentStep := 7; END_IF;
(* Rung 9: Step2 - Stopped If stop pressed / Step6 - Hold if hold pressed *)
IF (A1_Control.CurrentStep = 5) AND A1_Control.StopSelect THEN A1_Control.CurrentStep := 8; END_IF;
(* Rung 10: Step2 - Stopped If stop pressed / Step6 - Hold if hold pressed *)
IF (A1_Control.CurrentStep = 8) OR (((A1_Control.CurrentStep = 7) OR (A1_Control.CurrentStep = 4) OR (A1_Control.CurrentStep = 6)) AND A1_Control.StopSelect) THEN
    A1_Control.CurrentStep := 2;
END_IF;

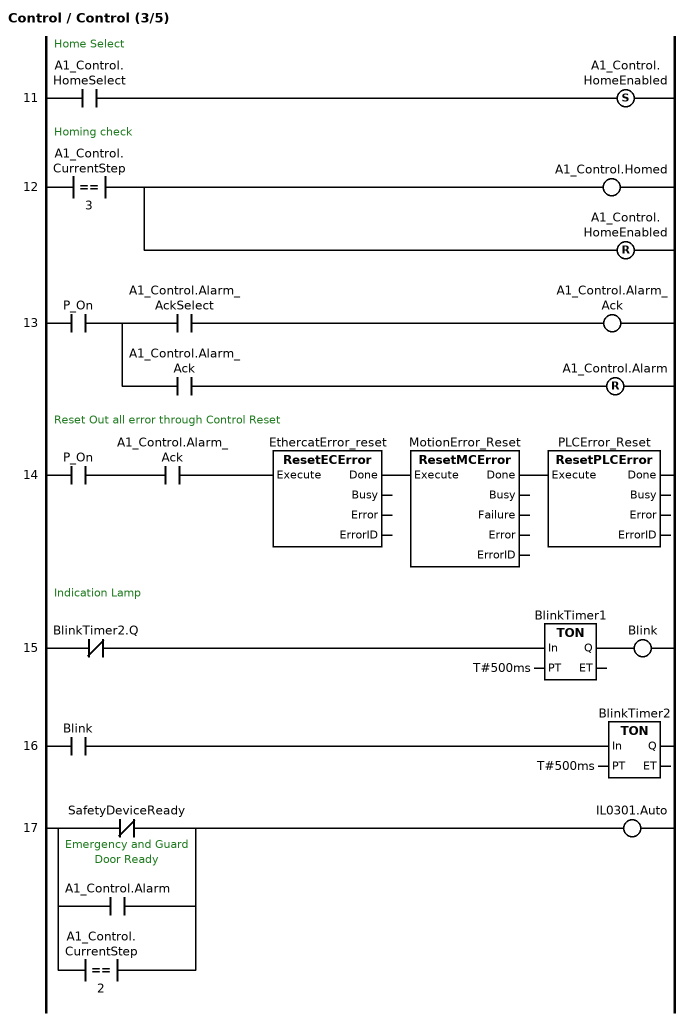
(* Rung 11: Home Select *)
IF A1_Control.HomeSelect THEN A1_Control.HomeEnabled := TRUE; END_IF;
(* Rung 12: Homing check *)
_p5 := A1_Control.CurrentStep = 3;
A1_Control.Homed := _p5;
IF _p5 THEN A1_Control.HomeEnabled := FALSE; END_IF;
(* Rung 13 *)
A1_Control.Alarm_Ack := P_On AND A1_Control.Alarm_AckSelect;
IF P_On AND A1_Control.Alarm_Ack THEN A1_Control.Alarm := FALSE; END_IF;
(* Rung 14: Reset Out all error through Control Reset *)
EthercatError_reset(Execute := P_On AND A1_Control.Alarm_Ack);
MotionError_Reset(Execute := EthercatError_reset.Done);
PLCError_Reset(Execute := MotionError_Reset.Done);
(* Rung 15: Indication Lamp *)
BlinkTimer1(In := NOT BlinkTimer2.Q, PT := T#500ms);
Blink := BlinkTimer1.Q;
(* Rung 16 *)
BlinkTimer2(In := Blink, PT := T#500ms);
(* Rung 17 *)
IL0301.Auto := NOT SafetyDeviceReady OR A1_Control.Alarm OR (A1_Control.CurrentStep = 2);

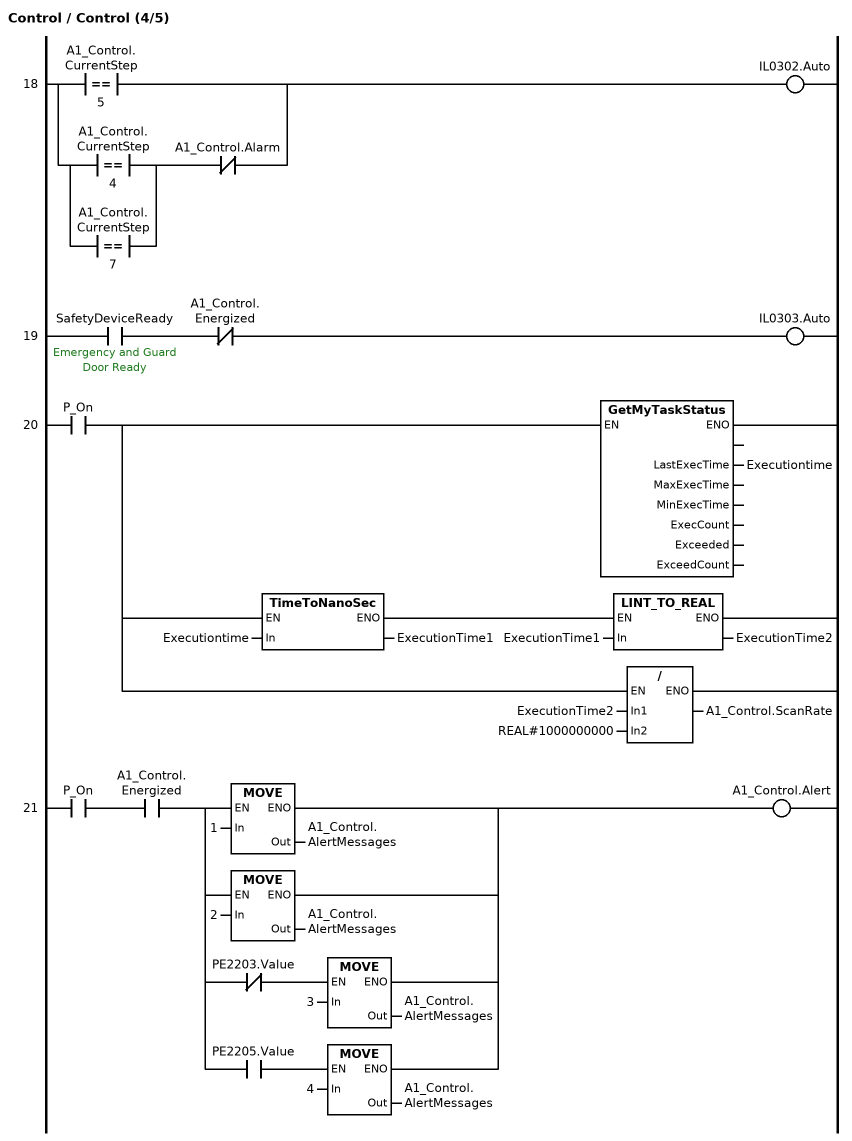
(* Rung 18 *)
IL0302.Auto := (A1_Control.CurrentStep = 5) OR (((A1_Control.CurrentStep = 4) OR (A1_Control.CurrentStep = 7)) AND NOT A1_Control.Alarm);
(* Rung 19 *)
IL0303.Auto := SafetyDeviceReady AND NOT A1_Control.Energized;
(* Rung 20 *)
IF P_On THEN
    GetMyTaskStatus(LastExecTime => Executiontime);
    ExecutionTime1 := TimeToNanoSec(In := Executiontime);
    ExecutionTime2 := LINT_TO_REAL(In := ExecutionTime1);
    A1_Control.ScanRate := ExecutionTime2 / REAL#1000000000;
END_IF;
(* Rung 21 *)
_p6 := P_On AND A1_Control.Energized;
IF _p6 THEN
    A1_Control.AlertMessages := 1;
    A1_Control.AlertMessages := 2;
END_IF;
IF _p6 AND NOT PE2203.Value THEN A1_Control.AlertMessages := 3; END_IF;
IF _p6 AND PE2205.Value THEN A1_Control.AlertMessages := 4; END_IF;
A1_Control.Alert := _p6 OR (_p6 AND (NOT PE2203.Value OR PE2205.Value));

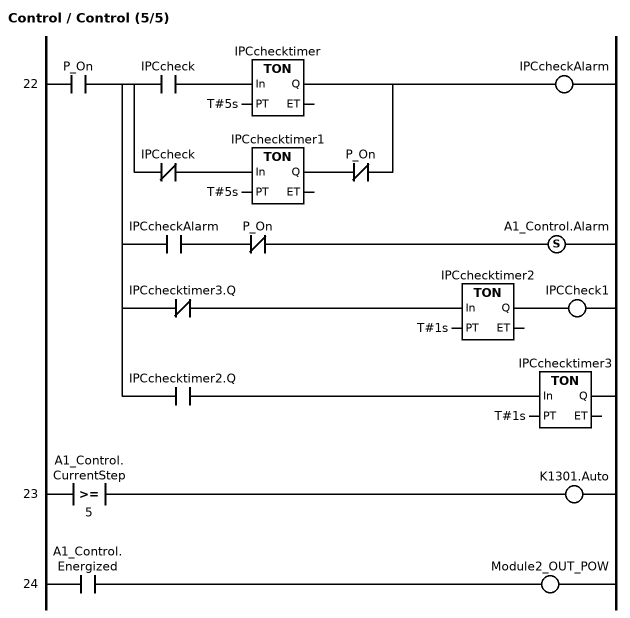
(* Rung 22 *)
IPCchecktimer(In := P_On AND IPCcheck, PT := T#5s);
IPCchecktimer1(In := P_On AND NOT IPCcheck, PT := T#5s);
IPCcheckAlarm := IPCchecktimer.Q OR (IPCchecktimer1.Q AND NOT P_On);
IF P_On AND IPCcheckAlarm AND NOT P_On THEN A1_Control.Alarm := TRUE; END_IF;
IPCchecktimer2(In := P_On AND NOT IPCchecktimer3.Q, PT := T#1s);
IPCCheck1 := IPCchecktimer2.Q;
IPCchecktimer3(In := P_On AND IPCchecktimer2.Q, PT := T#1s);
(* Rung 23 *)
K1301.Auto := A1_Control.CurrentStep >= 5;
(* Rung 24 *)
Module2_OUT_POW := A1_Control.Energized;

(* Section P14_Magazine: ladder, written here as Structured Text *)

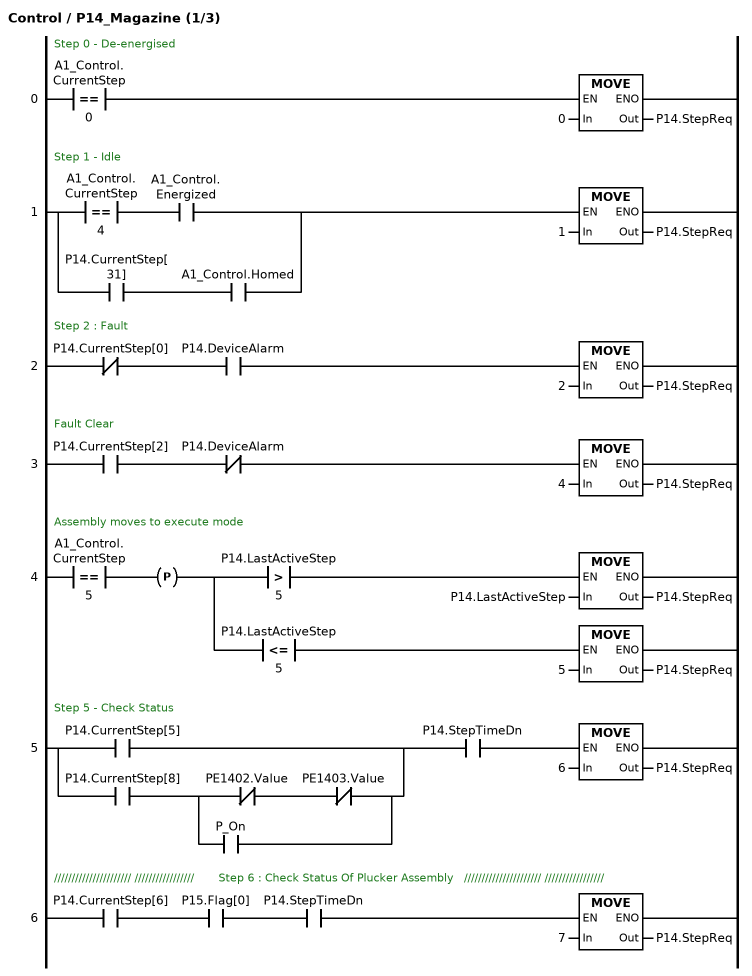
(* Rung 0: Step 0 - De-energised *)
IF A1_Control.CurrentStep = 0 THEN P14.StepReq := 0; END_IF;
(* Rung 1: Step 1 - Idle *)
IF ((A1_Control.CurrentStep = 4) AND A1_Control.Energized) OR (P14.CurrentStep[31] AND A1_Control.Homed) THEN
    P14.StepReq := 1;
END_IF;
(* Rung 2: Step 2 : Fault *)
IF NOT P14.CurrentStep[0] AND P14.DeviceAlarm THEN P14.StepReq := 2; END_IF;
(* Rung 3: Fault Clear *)
IF P14.CurrentStep[2] AND NOT P14.DeviceAlarm THEN P14.StepReq := 4; END_IF;
(* Rung 4: Assembly moves to execute mode *)
_e7(CLK := A1_Control.CurrentStep = 5);
IF _e7.Q AND (P14.LastActiveStep > 5) THEN P14.StepReq := P14.LastActiveStep; END_IF;
IF _e7.Q AND (P14.LastActiveStep <= 5) THEN P14.StepReq := 5; END_IF;
(* Rung 5: Step 5 - Check Status *)
IF (P14.CurrentStep[5] OR (P14.CurrentStep[8] AND ((NOT PE1402.Value AND NOT PE1403.Value) OR P_On))) AND P14.StepTimeDn THEN
    P14.StepReq := 6;
END_IF;
(* Rung 6: ////////////////////// /////////////////       Step 6 : Check Status Of Plucker Assembly   ////////////////////// ///////////////// *)
IF P14.CurrentStep[6] AND P15.Flag[0] AND P14.StepTimeDn THEN P14.StepReq := 7; END_IF;

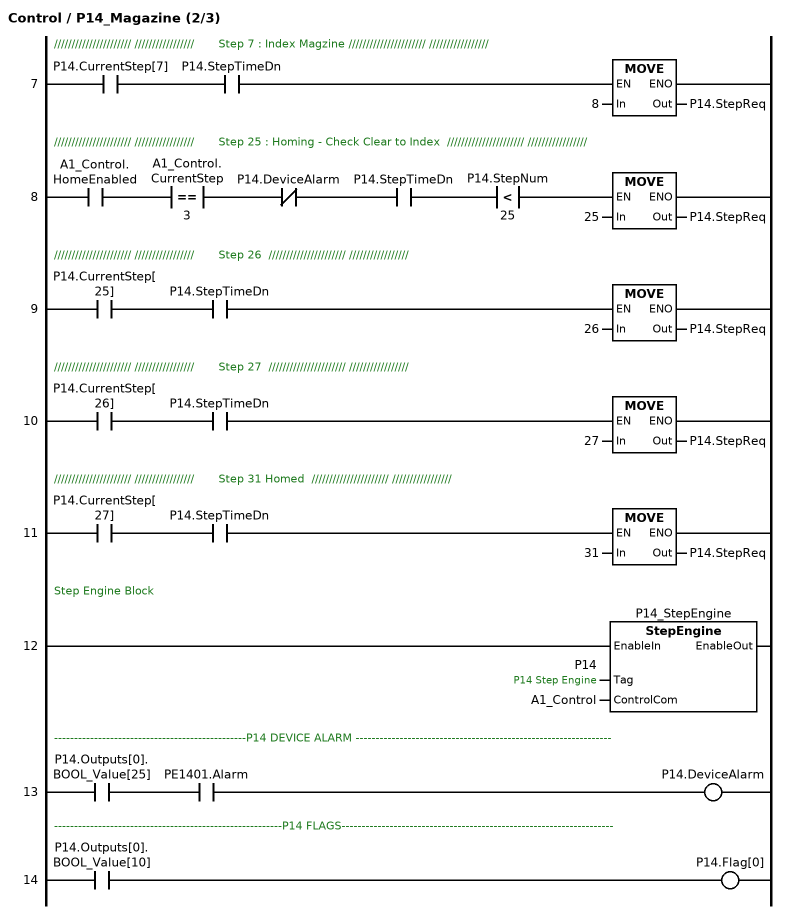
(* Rung 7: ////////////////////// /////////////////       Step 7 : Index Magzine ////////////////////// ///////////////// *)
IF P14.CurrentStep[7] AND P14.StepTimeDn THEN P14.StepReq := 8; END_IF;
(* Rung 8: ////////////////////// /////////////////       Step 25 : Homing - Check Clear to Index  ////////////////////// ///////////////// *)
IF A1_Control.HomeEnabled AND (A1_Control.CurrentStep = 3) AND NOT P14.DeviceAlarm AND P14.StepTimeDn AND (P14.StepNum < 25) THEN
    P14.StepReq := 25;
END_IF;
(* Rung 9: ////////////////////// /////////////////       Step 26  ////////////////////// ///////////////// *)
IF P14.CurrentStep[25] AND P14.StepTimeDn THEN P14.StepReq := 26; END_IF;
(* Rung 10: ////////////////////// /////////////////       Step 27  ////////////////////// ///////////////// *)
IF P14.CurrentStep[26] AND P14.StepTimeDn THEN P14.StepReq := 27; END_IF;
(* Rung 11: ////////////////////// /////////////////       Step 31 Homed  ////////////////////// ///////////////// *)
IF P14.CurrentStep[27] AND P14.StepTimeDn THEN P14.StepReq := 31; END_IF;
(* Rung 12: Step Engine Block *)
P14_StepEngine(EnableIn := TRUE, Tag := P14, ControlCom := A1_Control);
(* Rung 13: ------------------------------------------------P14 DEVICE ALARM ---------------------------------------------------------------- *)
P14.DeviceAlarm := P14.Outputs[0].BOOL_Value[25] AND PE1401.Alarm;
(* Rung 14: ---------------------------------------------------------P14 FLAGS-------------------------------------------------------------------- *)
P14.Flag[0] := P14.Outputs[0].BOOL_Value[10];

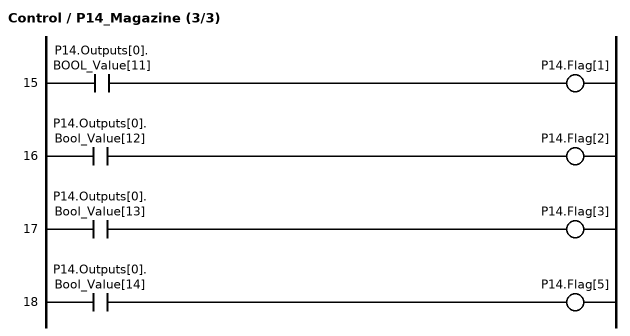
(* Rung 15 *)
P14.Flag[1] := P14.Outputs[0].BOOL_Value[11];
(* Rung 16 *)
P14.Flag[2] := P14.Outputs[0].Bool_Value[12];
(* Rung 17 *)
P14.Flag[3] := P14.Outputs[0].Bool_Value[13];
(* Rung 18 *)
P14.Flag[5] := P14.Outputs[0].Bool_Value[14];

(* Section P15_CaseErector: ladder, written here as Structured Text *)

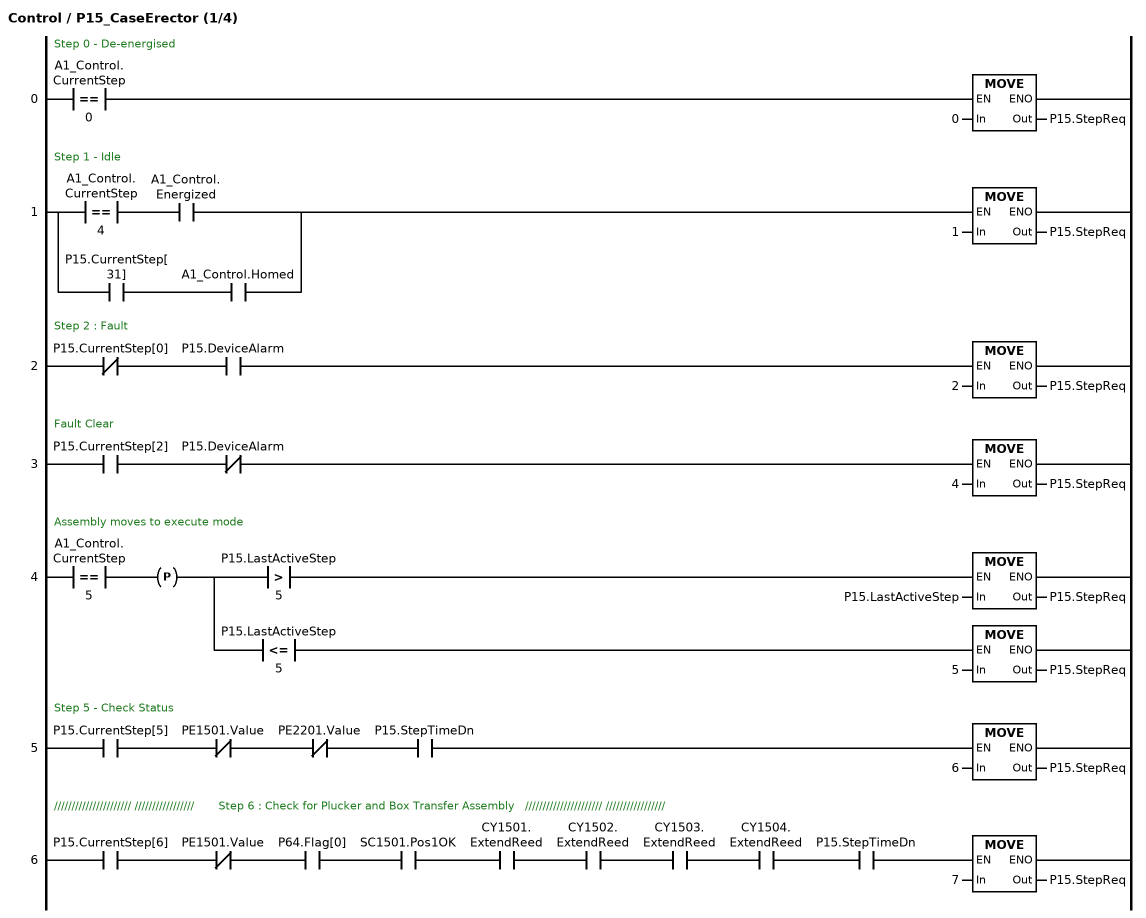
(* Rung 0: Step 0 - De-energised *)
IF A1_Control.CurrentStep = 0 THEN P15.StepReq := 0; END_IF;
(* Rung 1: Step 1 - Idle *)
IF ((A1_Control.CurrentStep = 4) AND A1_Control.Energized) OR (P15.CurrentStep[31] AND A1_Control.Homed) THEN
    P15.StepReq := 1;
END_IF;
(* Rung 2: Step 2 : Fault *)
IF NOT P15.CurrentStep[0] AND P15.DeviceAlarm THEN P15.StepReq := 2; END_IF;
(* Rung 3: Fault Clear *)
IF P15.CurrentStep[2] AND NOT P15.DeviceAlarm THEN P15.StepReq := 4; END_IF;
(* Rung 4: Assembly moves to execute mode *)
_e8(CLK := A1_Control.CurrentStep = 5);
IF _e8.Q AND (P15.LastActiveStep > 5) THEN P15.StepReq := P15.LastActiveStep; END_IF;
IF _e8.Q AND (P15.LastActiveStep <= 5) THEN P15.StepReq := 5; END_IF;
(* Rung 5: Step 5 - Check Status *)
IF P15.CurrentStep[5] AND NOT PE1501.Value AND NOT PE2201.Value AND P15.StepTimeDn THEN
    P15.StepReq := 6;
END_IF;
(* Rung 6: ////////////////////// /////////////////       Step 6 : Check for Plucker and Box Transfer Assembly   ////////////////////// ///////////////// *)
IF P15.CurrentStep[6] AND NOT PE1501.Value AND P64.Flag[0] AND SC1501.Pos1OK AND CY1501.ExtendReed AND CY1502.ExtendReed AND CY1503.ExtendReed AND CY1504.ExtendReed AND P15.StepTimeDn THEN
    P15.StepReq := 7;
END_IF;
(* notes on elements: Plucker Initial Pos *)

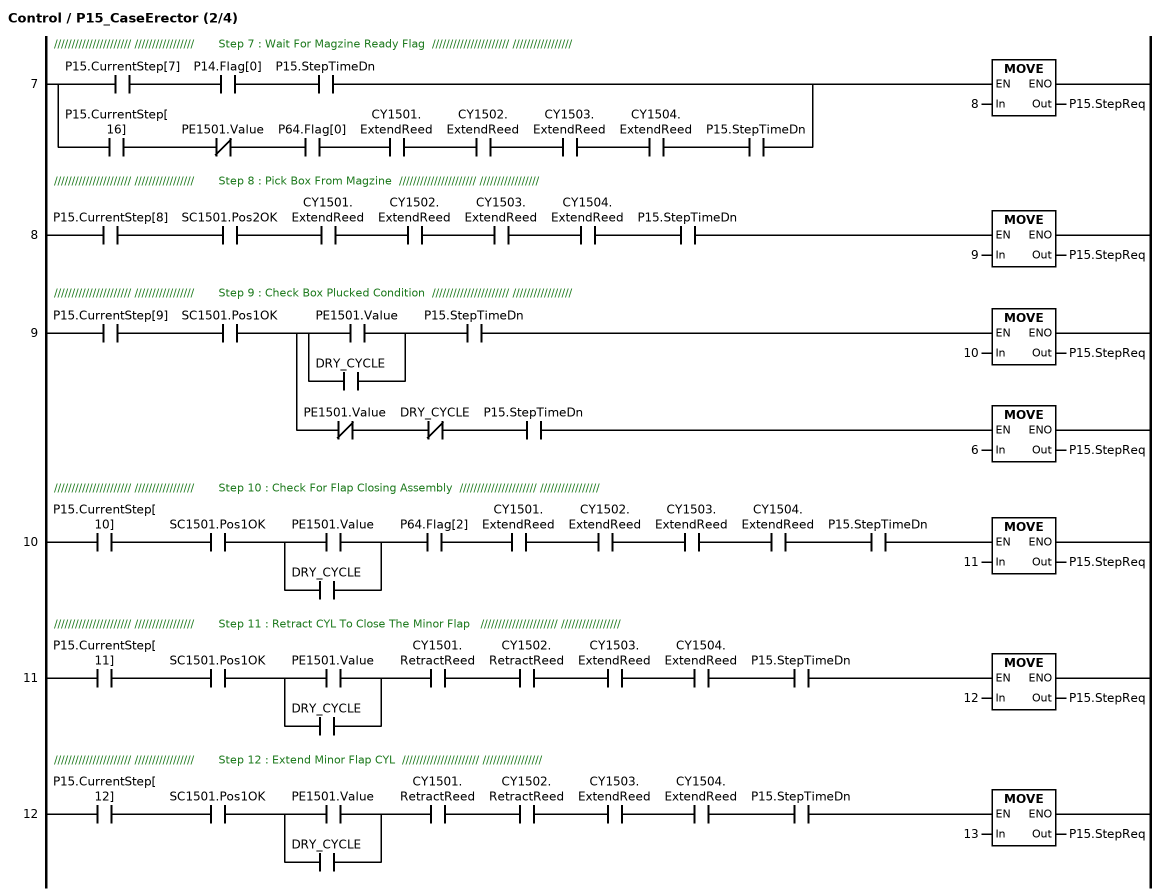
(* Rung 7: ////////////////////// /////////////////       Step 7 : Wait For Magzine Ready Flag  ////////////////////// ///////////////// *)
IF (P15.CurrentStep[7] AND P14.Flag[0] AND P15.StepTimeDn) OR (P15.CurrentStep[16] AND NOT PE1501.Value AND P64.Flag[0] AND CY1501.ExtendReed AND CY1502.ExtendReed AND CY1503.ExtendReed AND CY1504.ExtendReed AND P15.StepTimeDn) THEN
    P15.StepReq := 8;
END_IF;
(* Rung 8: ////////////////////// /////////////////       Step 8 : Pick Box From Magzine  ////////////////////// ///////////////// *)
IF P15.CurrentStep[8] AND SC1501.Pos2OK AND CY1501.ExtendReed AND CY1502.ExtendReed AND CY1503.ExtendReed AND CY1504.ExtendReed AND P15.StepTimeDn THEN
    P15.StepReq := 9;
END_IF;
(* notes on elements: Plucker Pluck Pos *)
(* Rung 9: ////////////////////// /////////////////       Step 9 : Check Box Plucked Condition  ////////////////////// ///////////////// *)
_p9 := P15.CurrentStep[9] AND SC1501.Pos1OK;
IF P15.CurrentStep[9] AND SC1501.Pos1OK AND (PE1501.Value OR DRY_CYCLE) AND P15.StepTimeDn THEN
    P15.StepReq := 10;
END_IF;
IF _p9 AND NOT PE1501.Value AND NOT DRY_CYCLE AND P15.StepTimeDn THEN P15.StepReq := 6; END_IF;
(* Rung 10: ////////////////////// /////////////////       Step 10 : Check For Flap Closing Assembly  ////////////////////// ///////////////// *)
IF P15.CurrentStep[10] AND SC1501.Pos1OK AND (PE1501.Value OR DRY_CYCLE) AND P64.Flag[2] AND CY1501.ExtendReed AND CY1502.ExtendReed AND CY1503.ExtendReed AND CY1504.ExtendReed AND P15.StepTimeDn THEN
    P15.StepReq := 11;
END_IF;
(* Rung 11: ////////////////////// /////////////////       Step 11 : Retract CYL To Close The Minor Flap   ////////////////////// ///////////////// *)
IF P15.CurrentStep[11] AND SC1501.Pos1OK AND (PE1501.Value OR DRY_CYCLE) AND CY1501.RetractReed AND CY1502.RetractReed AND CY1503.ExtendReed AND CY1504.ExtendReed AND P15.StepTimeDn THEN
    P15.StepReq := 12;
END_IF;
(* Rung 12: ////////////////////// /////////////////       Step 12 : Extend Minor Flap CYL  ////////////////////// ///////////////// *)
IF P15.CurrentStep[12] AND SC1501.Pos1OK AND (PE1501.Value OR DRY_CYCLE) AND CY1501.RetractReed AND CY1502.RetractReed AND CY1503.ExtendReed AND CY1504.ExtendReed AND P15.StepTimeDn THEN
    P15.StepReq := 13;
END_IF;

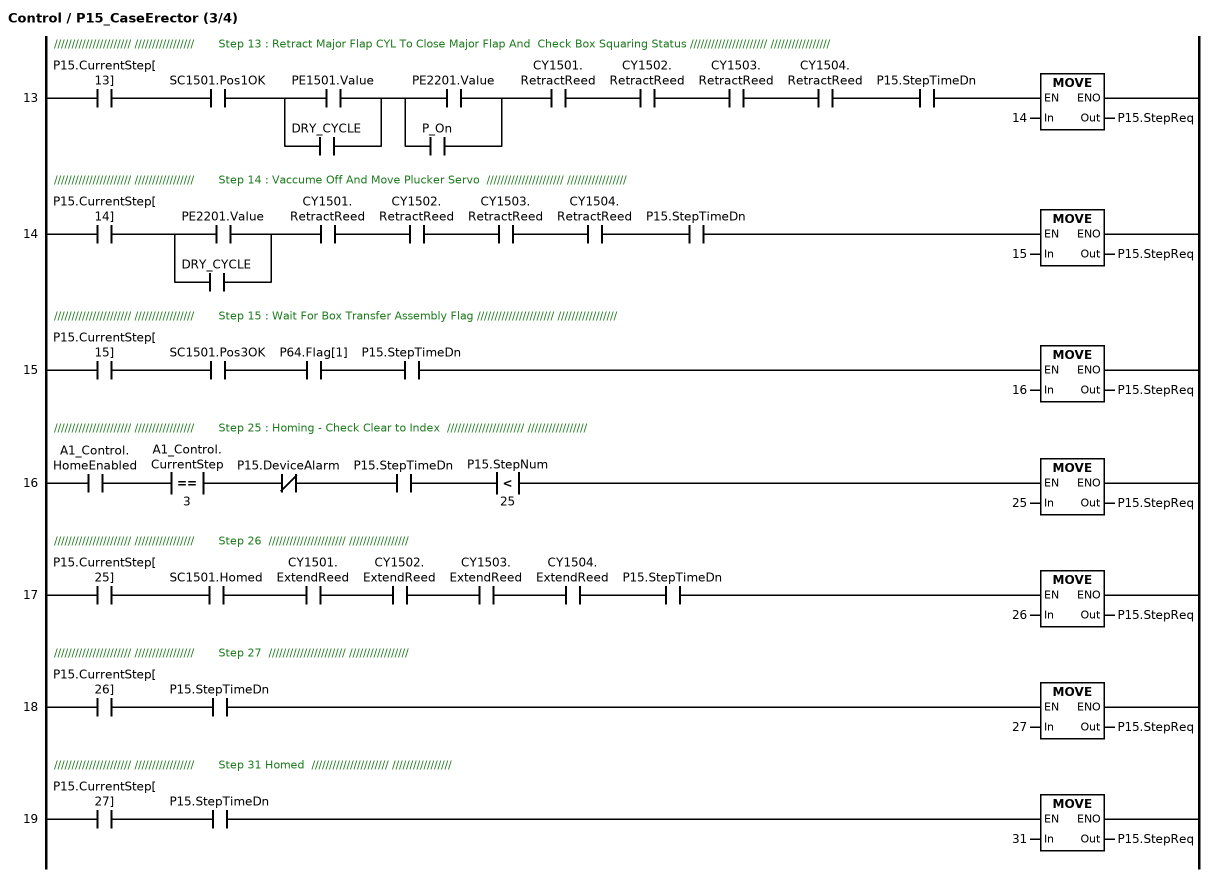
(* Rung 13: ////////////////////// /////////////////       Step 13 : Retract Major Flap CYL To Close Major Flap And  Check Box Squaring Status ////////////////////// ///////////////// *)
IF P15.CurrentStep[13] AND SC1501.Pos1OK AND (PE1501.Value OR DRY_CYCLE) AND (PE2201.Value OR P_On) AND CY1501.RetractReed AND CY1502.RetractReed AND CY1503.RetractReed AND CY1504.RetractReed AND P15.StepTimeDn THEN
    P15.StepReq := 14;
END_IF;
(* Rung 14: ////////////////////// /////////////////       Step 14 : Vaccume Off And Move Plucker Servo  ////////////////////// ///////////////// *)
IF P15.CurrentStep[14] AND (PE2201.Value OR DRY_CYCLE) AND CY1501.RetractReed AND CY1502.RetractReed AND CY1503.RetractReed AND CY1504.RetractReed AND P15.StepTimeDn THEN
    P15.StepReq := 15;
END_IF;
(* Rung 15: ////////////////////// /////////////////       Step 15 : Wait For Box Transfer Assembly Flag ////////////////////// ///////////////// *)
IF P15.CurrentStep[15] AND SC1501.Pos3OK AND P64.Flag[1] AND P15.StepTimeDn THEN
    P15.StepReq := 16;
END_IF;
(* Rung 16: ////////////////////// /////////////////       Step 25 : Homing - Check Clear to Index  ////////////////////// ///////////////// *)
IF A1_Control.HomeEnabled AND (A1_Control.CurrentStep = 3) AND NOT P15.DeviceAlarm AND P15.StepTimeDn AND (P15.StepNum < 25) THEN
    P15.StepReq := 25;
END_IF;
(* Rung 17: ////////////////////// /////////////////       Step 26  ////////////////////// ///////////////// *)
IF P15.CurrentStep[25] AND SC1501.Homed AND CY1501.ExtendReed AND CY1502.ExtendReed AND CY1503.ExtendReed AND CY1504.ExtendReed AND P15.StepTimeDn THEN
    P15.StepReq := 26;
END_IF;
(* Rung 18: ////////////////////// /////////////////       Step 27  ////////////////////// ///////////////// *)
IF P15.CurrentStep[26] AND P15.StepTimeDn THEN P15.StepReq := 27; END_IF;
(* Rung 19: ////////////////////// /////////////////       Step 31 Homed  ////////////////////// ///////////////// *)
IF P15.CurrentStep[27] AND P15.StepTimeDn THEN P15.StepReq := 31; END_IF;

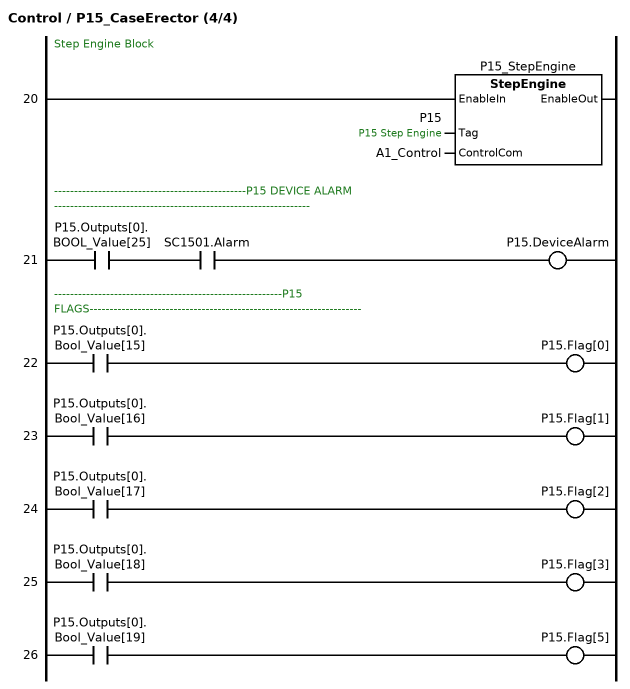
(* Rung 20: Step Engine Block *)
P15_StepEngine(EnableIn := TRUE, Tag := P15, ControlCom := A1_Control);
(* Rung 21: ------------------------------------------------P15 DEVICE ALARM ---------------------------------------------------------------- *)
P15.DeviceAlarm := P15.Outputs[0].BOOL_Value[25] AND SC1501.Alarm;
(* Rung 22: ---------------------------------------------------------P15 FLAGS-------------------------------------------------------------------- *)
P15.Flag[0] := P15.Outputs[0].Bool_Value[15];
(* Rung 23 *)
P15.Flag[1] := P15.Outputs[0].Bool_Value[16];
(* Rung 24 *)
P15.Flag[2] := P15.Outputs[0].Bool_Value[17];
(* Rung 25 *)
P15.Flag[3] := P15.Outputs[0].Bool_Value[18];
(* Rung 26 *)
P15.Flag[5] := P15.Outputs[0].Bool_Value[19];

(* Section P64_CaseTransfer: ladder, written here as Structured Text *)

